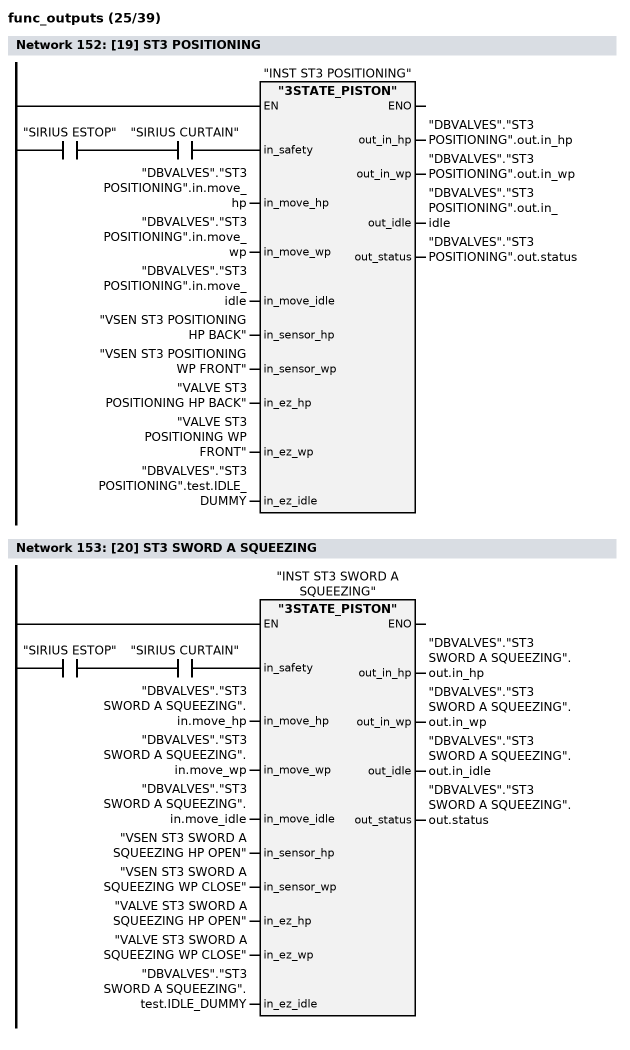
   RUNG wire#powerrail
      "INST ST3 POSITIONING"(in_safety := wire#w1, in_move_hp := "DBVALVES"."ST3 POSITIONING".in.move_hp, in_move_wp := "DBVALVES"."ST3 POSITIONING".in.move_wp, in_move_idle := "DBVALVES"."ST3 POSITIONING".in.move_idle, in_sensor_hp := "VSEN ST3 POSITIONING HP BACK", in_sensor_wp := "VSEN ST3 POSITIONING WP FRONT", in_ez_hp := "VALVE ST3 POSITIONING HP BACK", in_ez_wp := "VALVE ST3 POSITIONING WP FRONT", in_ez_idle := "DBVALVES"."ST3 POSITIONING".test.IDLE_DUMMY, out_in_hp => "DBVALVES"."ST3 POSITIONING".out.in_hp, out_in_wp => "DBVALVES"."ST3 POSITIONING".out.in_wp, out_idle => "DBVALVES"."ST3 POSITIONING".out.in_idle, out_status => "DBVALVES"."ST3 POSITIONING".out.status)
   END_RUNG
   RUNG wire#powerrail
      Contact( "SIRIUS ESTOP" )
      Contact( "SIRIUS CURTAIN" )
   END_RUNG wire#w1
   // the same network as SCL:
   "INST ST3 POSITIONING"(in_safety := "SIRIUS ESTOP" AND "SIRIUS CURTAIN",   // "3STATE_PISTON"
                          in_move_hp := "DBVALVES"."ST3 POSITIONING".in.move_hp,
                          in_move_wp := "DBVALVES"."ST3 POSITIONING".in.move_wp,
                          in_move_idle := "DBVALVES"."ST3 POSITIONING".in.move_idle,
                          in_sensor_hp := "VSEN ST3 POSITIONING HP BACK",
                          in_sensor_wp := "VSEN ST3 POSITIONING WP FRONT",
                          in_ez_hp := "VALVE ST3 POSITIONING HP BACK",
                          in_ez_wp := "VALVE ST3 POSITIONING WP FRONT",
                          in_ez_idle := "DBVALVES"."ST3 POSITIONING".test.IDLE_DUMMY,
                          out_in_hp => "DBVALVES"."ST3 POSITIONING".out.in_hp,
                          out_in_wp => "DBVALVES"."ST3 POSITIONING".out.in_wp,
                          out_idle => "DBVALVES"."ST3 POSITIONING".out.in_idle,
                          out_status => "DBVALVES"."ST3 POSITIONING".out.status);
END_REGION

REGION Network 153: [20] ST3 SWORD A SQUEEZING
   RUNG wire#powerrail
      "INST ST3 SWORD A SQUEEZING"(in_safety := wire#w1, in_move_hp := "DBVALVES"."ST3 SWORD A SQUEEZING".in.move_hp, in_move_wp := "DBVALVES"."ST3 SWORD A SQUEEZING".in.move_wp, in_move_idle := "DBVALVES"."ST3 SWORD A SQUEEZING".in.move_idle, in_sensor_hp := "VSEN ST3 SWORD A SQUEEZING HP OPEN", in_sensor_wp := "VSEN ST3 SWORD A SQUEEZING WP CLOSE", in_ez_hp := "VALVE ST3 SWORD A SQUEEZING HP OPEN", in_ez_wp := "VALVE ST3 SWORD A SQUEEZING WP CLOSE", in_ez_idle := "DBVALVES"."ST3 SWORD A SQUEEZING".test.IDLE_DUMMY, out_in_hp => "DBVALVES"."ST3 SWORD A SQUEEZING".out.in_hp, out_in_wp => "DBVALVES"."ST3 SWORD A SQUEEZING".out.in_wp, out_idle => "DBVALVES"."ST3 SWORD A SQUEEZING".out.in_idle, out_status => "DBVALVES"."ST3 SWORD A SQUEEZING".out.status)
   END_RUNG
   RUNG wire#powerrail
      Contact( "SIRIUS ESTOP" )
      Contact( "SIRIUS CURTAIN" )
   END_RUNG wire#w1
   // the same network as SCL:
   "INST ST3 SWORD A SQUEEZING"(in_safety := "SIRIUS ESTOP" AND "SIRIUS CURTAIN",   // "3STATE_PISTON"
                           in_move_hp := "DBVALVES"."ST3 SWORD A SQUEEZING".in.move_hp,
                           in_move_wp := "DBVALVES"."ST3 SWORD A SQUEEZING".in.move_wp,
                           in_move_idle := "DBVALVES"."ST3 SWORD A SQUEEZING".in.move_idle,
                           in_sensor_hp := "VSEN ST3 SWORD A SQUEEZING HP OPEN",
                           in_sensor_wp := "VSEN ST3 SWORD A SQUEEZING WP CLOSE",
                           in_ez_hp := "VALVE ST3 SWORD A SQUEEZING HP OPEN",
                           in_ez_wp := "VALVE ST3 SWORD A SQUEEZING WP CLOSE",
                           in_ez_idle := "DBVALVES"."ST3 SWORD A SQUEEZING".test.IDLE_DUMMY,
                           out_in_hp => "DBVALVES"."ST3 SWORD A SQUEEZING".out.in_hp,
                           out_in_wp => "DBVALVES"."ST3 SWORD A SQUEEZING".out.in_wp,
                           out_idle => "DBVALVES"."ST3 SWORD A SQUEEZING".out.in_idle,
                           out_status => "DBVALVES"."ST3 SWORD A SQUEEZING".out.status);
END_REGION

REGION Network 154: [21] ST3 SWORD A SPREADING
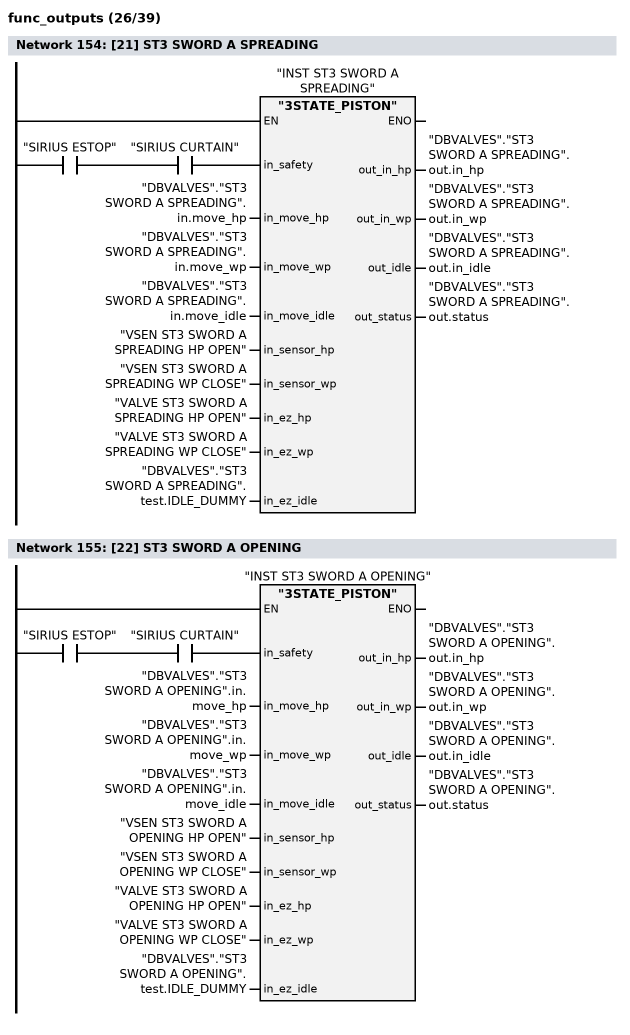
   RUNG wire#powerrail
      "INST ST3 SWORD A SPREADING"(in_safety := wire#w1, in_move_hp := "DBVALVES"."ST3 SWORD A SPREADING".in.move_hp, in_move_wp := "DBVALVES"."ST3 SWORD A SPREADING".in.move_wp, in_move_idle := "DBVALVES"."ST3 SWORD A SPREADING".in.move_idle, in_sensor_hp := "VSEN ST3 SWORD A SPREADING HP OPEN", in_sensor_wp := "VSEN ST3 SWORD A SPREADING WP CLOSE", in_ez_hp := "VALVE ST3 SWORD A SPREADING HP OPEN", in_ez_wp := "VALVE ST3 SWORD A SPREADING WP CLOSE", in_ez_idle := "DBVALVES"."ST3 SWORD A SPREADING".test.IDLE_DUMMY, out_in_hp => "DBVALVES"."ST3 SWORD A SPREADING".out.in_hp, out_in_wp => "DBVALVES"."ST3 SWORD A SPREADING".out.in_wp, out_idle => "DBVALVES"."ST3 SWORD A SPREADING".out.in_idle, out_status => "DBVALVES"."ST3 SWORD A SPREADING".out.status)
   END_RUNG
   RUNG wire#powerrail
      Contact( "SIRIUS ESTOP" )
      Contact( "SIRIUS CURTAIN" )
   END_RUNG wire#w1
   // the same network as SCL:
   "INST ST3 SWORD A SPREADING"(in_safety := "SIRIUS ESTOP" AND "SIRIUS CURTAIN",   // "3STATE_PISTON"
                           in_move_hp := "DBVALVES"."ST3 SWORD A SPREADING".in.move_hp,
                           in_move_wp := "DBVALVES"."ST3 SWORD A SPREADING".in.move_wp,
                           in_move_idle := "DBVALVES"."ST3 SWORD A SPREADING".in.move_idle,
                           in_sensor_hp := "VSEN ST3 SWORD A SPREADING HP OPEN",
                           in_sensor_wp := "VSEN ST3 SWORD A SPREADING WP CLOSE",
                           in_ez_hp := "VALVE ST3 SWORD A SPREADING HP OPEN",
                           in_ez_wp := "VALVE ST3 SWORD A SPREADING WP CLOSE",
                           in_ez_idle := "DBVALVES"."ST3 SWORD A SPREADING".test.IDLE_DUMMY,
                           out_in_hp => "DBVALVES"."ST3 SWORD A SPREADING".out.in_hp,
                           out_in_wp => "DBVALVES"."ST3 SWORD A SPREADING".out.in_wp,
                           out_idle => "DBVALVES"."ST3 SWORD A SPREADING".out.in_idle,
                           out_status => "DBVALVES"."ST3 SWORD A SPREADING".out.status);
END_REGION

REGION Network 155: [22] ST3 SWORD A OPENING
   RUNG wire#powerrail
      "INST ST3 SWORD A OPENING"(in_safety := wire#w1, in_move_hp := "DBVALVES"."ST3 SWORD A OPENING".in.move_hp, in_move_wp := "DBVALVES"."ST3 SWORD A OPENING".in.move_wp, in_move_idle := "DBVALVES"."ST3 SWORD A OPENING".in.move_idle, in_sensor_hp := "VSEN ST3 SWORD A OPENING HP OPEN", in_sensor_wp := "VSEN ST3 SWORD A OPENING WP CLOSE", in_ez_hp := "VALVE ST3 SWORD A OPENING HP OPEN", in_ez_wp := "VALVE ST3 SWORD A OPENING WP CLOSE", in_ez_idle := "DBVALVES"."ST3 SWORD A OPENING".test.IDLE_DUMMY, out_in_hp => "DBVALVES"."ST3 SWORD A OPENING".out.in_hp, out_in_wp => "DBVALVES"."ST3 SWORD A OPENING".out.in_wp, out_idle => "DBVALVES"."ST3 SWORD A OPENING".out.in_idle, out_status => "DBVALVES"."ST3 SWORD A OPENING".out.status)
   END_RUNG
   RUNG wire#powerrail
      Contact( "SIRIUS ESTOP" )
      Contact( "SIRIUS CURTAIN" )
   END_RUNG wire#w1
   // the same network as SCL:
   "INST ST3 SWORD A OPENING"(in_safety := "SIRIUS ESTOP" AND "SIRIUS CURTAIN",   // "3STATE_PISTON"
                           in_move_hp := "DBVALVES"."ST3 SWORD A OPENING".in.move_hp,
                           in_move_wp := "DBVALVES"."ST3 SWORD A OPENING".in.move_wp,
                           in_move_idle := "DBVALVES"."ST3 SWORD A OPENING".in.move_idle,
                           in_sensor_hp := "VSEN ST3 SWORD A OPENING HP OPEN",
                           in_sensor_wp := "VSEN ST3 SWORD A OPENING WP CLOSE",
                           in_ez_hp := "VALVE ST3 SWORD A OPENING HP OPEN",
                           in_ez_wp := "VALVE ST3 SWORD A OPENING WP CLOSE",
                           in_ez_idle := "DBVALVES"."ST3 SWORD A OPENING".test.IDLE_DUMMY,
                           out_in_hp => "DBVALVES"."ST3 SWORD A OPENING".out.in_hp,
                           out_in_wp => "DBVALVES"."ST3 SWORD A OPENING".out.in_wp,
                           out_idle => "DBVALVES"."ST3 SWORD A OPENING".out.in_idle,
                           out_status => "DBVALVES"."ST3 SWORD A OPENING".out.status);
END_REGION

REGION Network 156: [23] ST3 SWORD B SQUEEZING
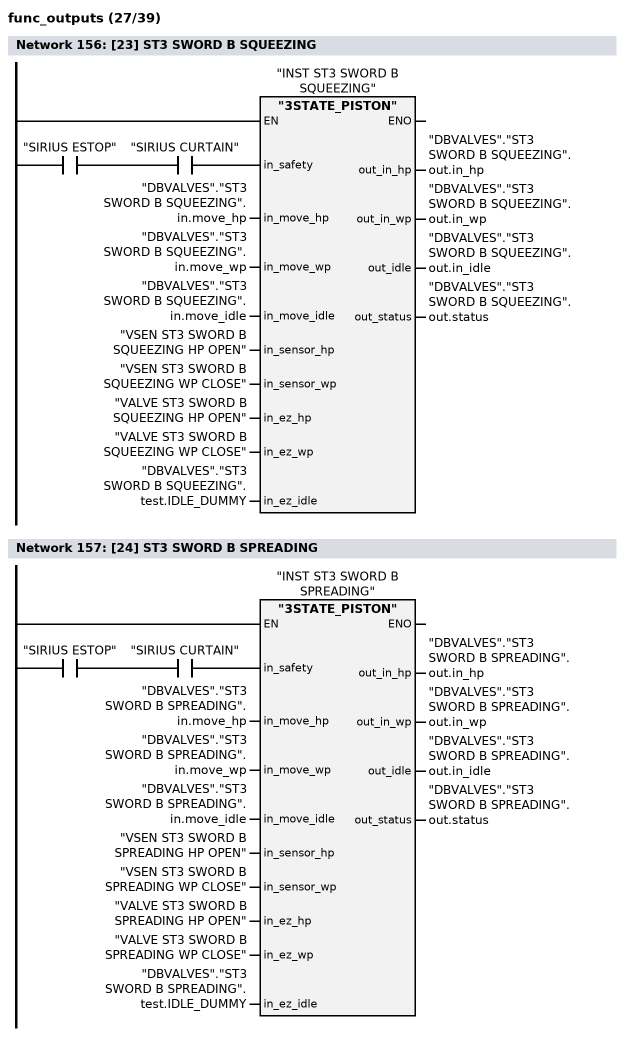
   RUNG wire#powerrail
      "INST ST3 SWORD B SQUEEZING"(in_safety := wire#w1, in_move_hp := "DBVALVES"."ST3 SWORD B SQUEEZING".in.move_hp, in_move_wp := "DBVALVES"."ST3 SWORD B SQUEEZING".in.move_wp, in_move_idle := "DBVALVES"."ST3 SWORD B SQUEEZING".in.move_idle, in_sensor_hp := "VSEN ST3 SWORD B SQUEEZING HP OPEN", in_sensor_wp := "VSEN ST3 SWORD B SQUEEZING WP CLOSE", in_ez_hp := "VALVE ST3 SWORD B SQUEEZING HP OPEN", in_ez_wp := "VALVE ST3 SWORD B SQUEEZING WP CLOSE", in_ez_idle := "DBVALVES"."ST3 SWORD B SQUEEZING".test.IDLE_DUMMY, out_in_hp => "DBVALVES"."ST3 SWORD B SQUEEZING".out.in_hp, out_in_wp => "DBVALVES"."ST3 SWORD B SQUEEZING".out.in_wp, out_idle => "DBVALVES"."ST3 SWORD B SQUEEZING".out.in_idle, out_status => "DBVALVES"."ST3 SWORD B SQUEEZING".out.status)
   END_RUNG
   RUNG wire#powerrail
      Contact( "SIRIUS ESTOP" )
      Contact( "SIRIUS CURTAIN" )
   END_RUNG wire#w1
   // the same network as SCL:
   "INST ST3 SWORD B SQUEEZING"(in_safety := "SIRIUS ESTOP" AND "SIRIUS CURTAIN",   // "3STATE_PISTON"
                           in_move_hp := "DBVALVES"."ST3 SWORD B SQUEEZING".in.move_hp,
                           in_move_wp := "DBVALVES"."ST3 SWORD B SQUEEZING".in.move_wp,
                           in_move_idle := "DBVALVES"."ST3 SWORD B SQUEEZING".in.move_idle,
                           in_sensor_hp := "VSEN ST3 SWORD B SQUEEZING HP OPEN",
                           in_sensor_wp := "VSEN ST3 SWORD B SQUEEZING WP CLOSE",
                           in_ez_hp := "VALVE ST3 SWORD B SQUEEZING HP OPEN",
                           in_ez_wp := "VALVE ST3 SWORD B SQUEEZING WP CLOSE",
                           in_ez_idle := "DBVALVES"."ST3 SWORD B SQUEEZING".test.IDLE_DUMMY,
                           out_in_hp => "DBVALVES"."ST3 SWORD B SQUEEZING".out.in_hp,
                           out_in_wp => "DBVALVES"."ST3 SWORD B SQUEEZING".out.in_wp,
                           out_idle => "DBVALVES"."ST3 SWORD B SQUEEZING".out.in_idle,
                           out_status => "DBVALVES"."ST3 SWORD B SQUEEZING".out.status);
END_REGION

REGION Network 157: [24] ST3 SWORD B SPREADING
   RUNG wire#powerrail
      "INST ST3 SWORD B SPREADING"(in_safety := wire#w1, in_move_hp := "DBVALVES"."ST3 SWORD B SPREADING".in.move_hp, in_move_wp := "DBVALVES"."ST3 SWORD B SPREADING".in.move_wp, in_move_idle := "DBVALVES"."ST3 SWORD B SPREADING".in.move_idle, in_sensor_hp := "VSEN ST3 SWORD B SPREADING HP OPEN", in_sensor_wp := "VSEN ST3 SWORD B SPREADING WP CLOSE", in_ez_hp := "VALVE ST3 SWORD B SPREADING HP OPEN", in_ez_wp := "VALVE ST3 SWORD B SPREADING WP CLOSE", in_ez_idle := "DBVALVES"."ST3 SWORD B SPREADING".test.IDLE_DUMMY, out_in_hp => "DBVALVES"."ST3 SWORD B SPREADING".out.in_hp, out_in_wp => "DBVALVES"."ST3 SWORD B SPREADING".out.in_wp, out_idle => "DBVALVES"."ST3 SWORD B SPREADING".out.in_idle, out_status => "DBVALVES"."ST3 SWORD B SPREADING".out.status)
   END_RUNG
   RUNG wire#powerrail
      Contact( "SIRIUS ESTOP" )
      Contact( "SIRIUS CURTAIN" )
   END_RUNG wire#w1
   // the same network as SCL:
   "INST ST3 SWORD B SPREADING"(in_safety := "SIRIUS ESTOP" AND "SIRIUS CURTAIN",   // "3STATE_PISTON"
                           in_move_hp := "DBVALVES"."ST3 SWORD B SPREADING".in.move_hp,
                           in_move_wp := "DBVALVES"."ST3 SWORD B SPREADING".in.move_wp,
                           in_move_idle := "DBVALVES"."ST3 SWORD B SPREADING".in.move_idle,
                           in_sensor_hp := "VSEN ST3 SWORD B SPREADING HP OPEN",
                           in_sensor_wp := "VSEN ST3 SWORD B SPREADING WP CLOSE",
                           in_ez_hp := "VALVE ST3 SWORD B SPREADING HP OPEN",
                           in_ez_wp := "VALVE ST3 SWORD B SPREADING WP CLOSE",
                           in_ez_idle := "DBVALVES"."ST3 SWORD B SPREADING".test.IDLE_DUMMY,
                           out_in_hp => "DBVALVES"."ST3 SWORD B SPREADING".out.in_hp,
                           out_in_wp => "DBVALVES"."ST3 SWORD B SPREADING".out.in_wp,
                           out_idle => "DBVALVES"."ST3 SWORD B SPREADING".out.in_idle,
                           out_status => "DBVALVES"."ST3 SWORD B SPREADING".out.status);
END_REGION

REGION Network 158: [25] ST3 SWORD B OPENING
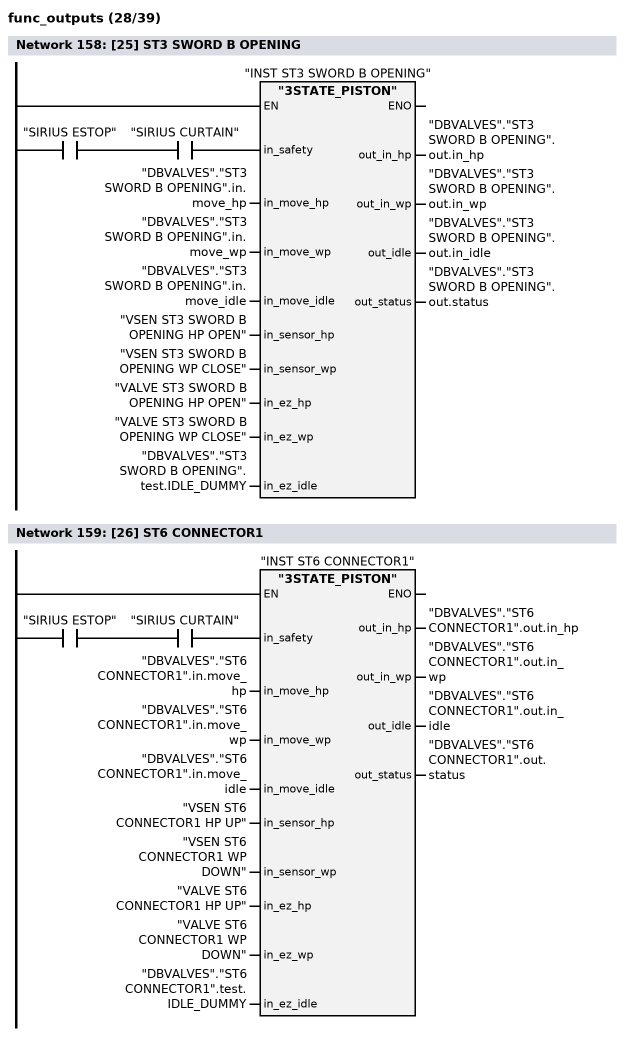
   RUNG wire#powerrail
      "INST ST3 SWORD B OPENING"(in_safety := wire#w1, in_move_hp := "DBVALVES"."ST3 SWORD B OPENING".in.move_hp, in_move_wp := "DBVALVES"."ST3 SWORD B OPENING".in.move_wp, in_move_idle := "DBVALVES"."ST3 SWORD B OPENING".in.move_idle, in_sensor_hp := "VSEN ST3 SWORD B OPENING HP OPEN", in_sensor_wp := "VSEN ST3 SWORD B OPENING WP CLOSE", in_ez_hp := "VALVE ST3 SWORD B OPENING HP OPEN", in_ez_wp := "VALVE ST3 SWORD B OPENING WP CLOSE", in_ez_idle := "DBVALVES"."ST3 SWORD B OPENING".test.IDLE_DUMMY, out_in_hp => "DBVALVES"."ST3 SWORD B OPENING".out.in_hp, out_in_wp => "DBVALVES"."ST3 SWORD B OPENING".out.in_wp, out_idle => "DBVALVES"."ST3 SWORD B OPENING".out.in_idle, out_status => "DBVALVES"."ST3 SWORD B OPENING".out.status)
   END_RUNG
   RUNG wire#powerrail
      Contact( "SIRIUS ESTOP" )
      Contact( "SIRIUS CURTAIN" )
   END_RUNG wire#w1
   // the same network as SCL:
   "INST ST3 SWORD B OPENING"(in_safety := "SIRIUS ESTOP" AND "SIRIUS CURTAIN",   // "3STATE_PISTON"
                           in_move_hp := "DBVALVES"."ST3 SWORD B OPENING".in.move_hp,
                           in_move_wp := "DBVALVES"."ST3 SWORD B OPENING".in.move_wp,
                           in_move_idle := "DBVALVES"."ST3 SWORD B OPENING".in.move_idle,
                           in_sensor_hp := "VSEN ST3 SWORD B OPENING HP OPEN",
                           in_sensor_wp := "VSEN ST3 SWORD B OPENING WP CLOSE",
                           in_ez_hp := "VALVE ST3 SWORD B OPENING HP OPEN",
                           in_ez_wp := "VALVE ST3 SWORD B OPENING WP CLOSE",
                           in_ez_idle := "DBVALVES"."ST3 SWORD B OPENING".test.IDLE_DUMMY,
                           out_in_hp => "DBVALVES"."ST3 SWORD B OPENING".out.in_hp,
                           out_in_wp => "DBVALVES"."ST3 SWORD B OPENING".out.in_wp,
                           out_idle => "DBVALVES"."ST3 SWORD B OPENING".out.in_idle,
                           out_status => "DBVALVES"."ST3 SWORD B OPENING".out.status);
END_REGION

REGION Network 159: [26] ST6 CONNECTOR1
   RUNG wire#powerrail
      "INST ST6 CONNECTOR1"(in_safety := wire#w1, in_move_hp := "DBVALVES"."ST6 CONNECTOR1".in.move_hp, in_move_wp := "DBVALVES"."ST6 CONNECTOR1".in.move_wp, in_move_idle := "DBVALVES"."ST6 CONNECTOR1".in.move_idle, in_sensor_hp := "VSEN ST6 CONNECTOR1 HP UP", in_sensor_wp := "VSEN ST6 CONNECTOR1 WP DOWN", in_ez_hp := "VALVE ST6 CONNECTOR1 HP UP", in_ez_wp := "VALVE ST6 CONNECTOR1 WP DOWN", in_ez_idle := "DBVALVES"."ST6 CONNECTOR1".test.IDLE_DUMMY, out_in_hp => "DBVALVES"."ST6 CONNECTOR1".out.in_hp, out_in_wp => "DBVALVES"."ST6 CONNECTOR1".out.in_wp, out_idle => "DBVALVES"."ST6 CONNECTOR1".out.in_idle, out_status => "DBVALVES"."ST6 CONNECTOR1".out.status)
   END_RUNG
   RUNG wire#powerrail
      Contact( "SIRIUS ESTOP" )
      Contact( "SIRIUS CURTAIN" )
   END_RUNG wire#w1
   // the same network as SCL:
   "INST ST6 CONNECTOR1"(in_safety := "SIRIUS ESTOP" AND "SIRIUS CURTAIN",   // "3STATE_PISTON"
                         in_move_hp := "DBVALVES"."ST6 CONNECTOR1".in.move_hp,
                         in_move_wp := "DBVALVES"."ST6 CONNECTOR1".in.move_wp,
                         in_move_idle := "DBVALVES"."ST6 CONNECTOR1".in.move_idle,
                         in_sensor_hp := "VSEN ST6 CONNECTOR1 HP UP",
                         in_sensor_wp := "VSEN ST6 CONNECTOR1 WP DOWN",
                         in_ez_hp := "VALVE ST6 CONNECTOR1 HP UP",
                         in_ez_wp := "VALVE ST6 CONNECTOR1 WP DOWN",
                         in_ez_idle := "DBVALVES"."ST6 CONNECTOR1".test.IDLE_DUMMY,
                         out_in_hp => "DBVALVES"."ST6 CONNECTOR1".out.in_hp,
                         out_in_wp => "DBVALVES"."ST6 CONNECTOR1".out.in_wp,
                         out_idle => "DBVALVES"."ST6 CONNECTOR1".out.in_idle,
                         out_status => "DBVALVES"."ST6 CONNECTOR1".out.status);
END_REGION

REGION Network 160: [27] ST6 CONNECTOR2
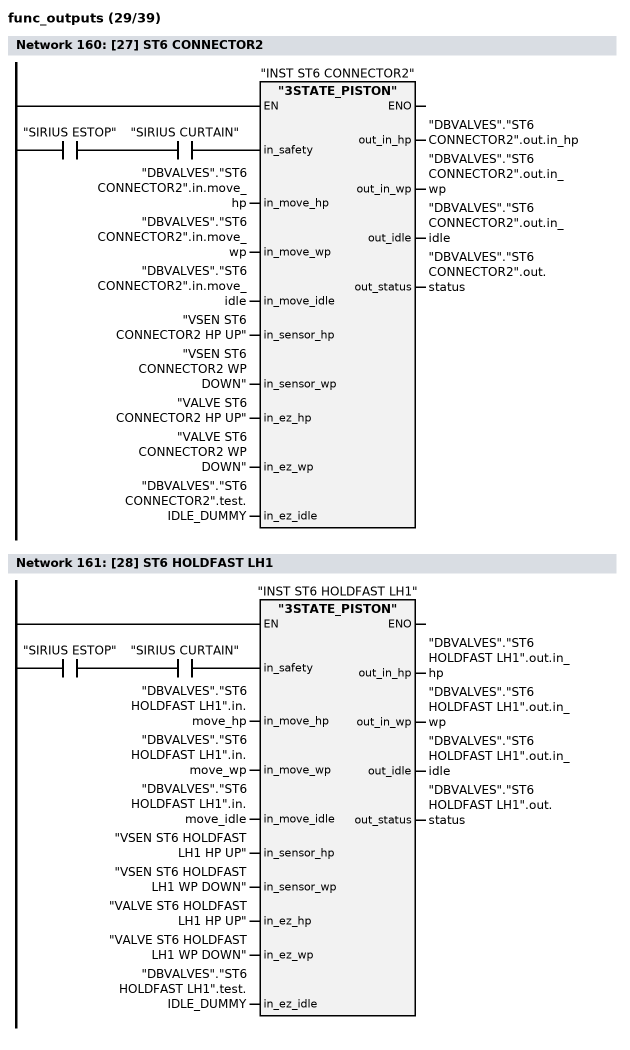
   RUNG wire#powerrail
      "INST ST6 CONNECTOR2"(in_safety := wire#w1, in_move_hp := "DBVALVES"."ST6 CONNECTOR2".in.move_hp, in_move_wp := "DBVALVES"."ST6 CONNECTOR2".in.move_wp, in_move_idle := "DBVALVES"."ST6 CONNECTOR2".in.move_idle, in_sensor_hp := "VSEN ST6 CONNECTOR2 HP UP", in_sensor_wp := "VSEN ST6 CONNECTOR2 WP DOWN", in_ez_hp := "VALVE ST6 CONNECTOR2 HP UP", in_ez_wp := "VALVE ST6 CONNECTOR2 WP DOWN", in_ez_idle := "DBVALVES"."ST6 CONNECTOR2".test.IDLE_DUMMY, out_in_hp => "DBVALVES"."ST6 CONNECTOR2".out.in_hp, out_in_wp => "DBVALVES"."ST6 CONNECTOR2".out.in_wp, out_idle => "DBVALVES"."ST6 CONNECTOR2".out.in_idle, out_status => "DBVALVES"."ST6 CONNECTOR2".out.status)
   END_RUNG
   RUNG wire#powerrail
      Contact( "SIRIUS ESTOP" )
      Contact( "SIRIUS CURTAIN" )
   END_RUNG wire#w1
   // the same network as SCL:
   "INST ST6 CONNECTOR2"(in_safety := "SIRIUS ESTOP" AND "SIRIUS CURTAIN",   // "3STATE_PISTON"
                         in_move_hp := "DBVALVES"."ST6 CONNECTOR2".in.move_hp,
                         in_move_wp := "DBVALVES"."ST6 CONNECTOR2".in.move_wp,
                         in_move_idle := "DBVALVES"."ST6 CONNECTOR2".in.move_idle,
                         in_sensor_hp := "VSEN ST6 CONNECTOR2 HP UP",
                         in_sensor_wp := "VSEN ST6 CONNECTOR2 WP DOWN",
                         in_ez_hp := "VALVE ST6 CONNECTOR2 HP UP",
                         in_ez_wp := "VALVE ST6 CONNECTOR2 WP DOWN",
                         in_ez_idle := "DBVALVES"."ST6 CONNECTOR2".test.IDLE_DUMMY,
                         out_in_hp => "DBVALVES"."ST6 CONNECTOR2".out.in_hp,
                         out_in_wp => "DBVALVES"."ST6 CONNECTOR2".out.in_wp,
                         out_idle => "DBVALVES"."ST6 CONNECTOR2".out.in_idle,
                         out_status => "DBVALVES"."ST6 CONNECTOR2".out.status);
END_REGION

REGION Network 161: [28] ST6 HOLDFAST LH1
   RUNG wire#powerrail
      "INST ST6 HOLDFAST LH1"(in_safety := wire#w1, in_move_hp := "DBVALVES"."ST6 HOLDFAST LH1".in.move_hp, in_move_wp := "DBVALVES"."ST6 HOLDFAST LH1".in.move_wp, in_move_idle := "DBVALVES"."ST6 HOLDFAST LH1".in.move_idle, in_sensor_hp := "VSEN ST6 HOLDFAST LH1 HP UP", in_sensor_wp := "VSEN ST6 HOLDFAST LH1 WP DOWN", in_ez_hp := "VALVE ST6 HOLDFAST LH1 HP UP", in_ez_wp := "VALVE ST6 HOLDFAST LH1 WP DOWN", in_ez_idle := "DBVALVES"."ST6 HOLDFAST LH1".test.IDLE_DUMMY, out_in_hp => "DBVALVES"."ST6 HOLDFAST LH1".out.in_hp, out_in_wp => "DBVALVES"."ST6 HOLDFAST LH1".out.in_wp, out_idle => "DBVALVES"."ST6 HOLDFAST LH1".out.in_idle, out_status => "DBVALVES"."ST6 HOLDFAST LH1".out.status)
   END_RUNG
   RUNG wire#powerrail
      Contact( "SIRIUS ESTOP" )
      Contact( "SIRIUS CURTAIN" )
   END_RUNG wire#w1
   // the same network as SCL:
   "INST ST6 HOLDFAST LH1"(in_safety := "SIRIUS ESTOP" AND "SIRIUS CURTAIN",   // "3STATE_PISTON"
                           in_move_hp := "DBVALVES"."ST6 HOLDFAST LH1".in.move_hp,
                           in_move_wp := "DBVALVES"."ST6 HOLDFAST LH1".in.move_wp,
                           in_move_idle := "DBVALVES"."ST6 HOLDFAST LH1".in.move_idle,
                           in_sensor_hp := "VSEN ST6 HOLDFAST LH1 HP UP",
                           in_sensor_wp := "VSEN ST6 HOLDFAST LH1 WP DOWN",
                           in_ez_hp := "VALVE ST6 HOLDFAST LH1 HP UP",
                           in_ez_wp := "VALVE ST6 HOLDFAST LH1 WP DOWN",
                           in_ez_idle := "DBVALVES"."ST6 HOLDFAST LH1".test.IDLE_DUMMY,
                           out_in_hp => "DBVALVES"."ST6 HOLDFAST LH1".out.in_hp,
                           out_in_wp => "DBVALVES"."ST6 HOLDFAST LH1".out.in_wp,
                           out_idle => "DBVALVES"."ST6 HOLDFAST LH1".out.in_idle,
                           out_status => "DBVALVES"."ST6 HOLDFAST LH1".out.status);
END_REGION

REGION Network 162: [29] ST6 HOLDFAST LH2
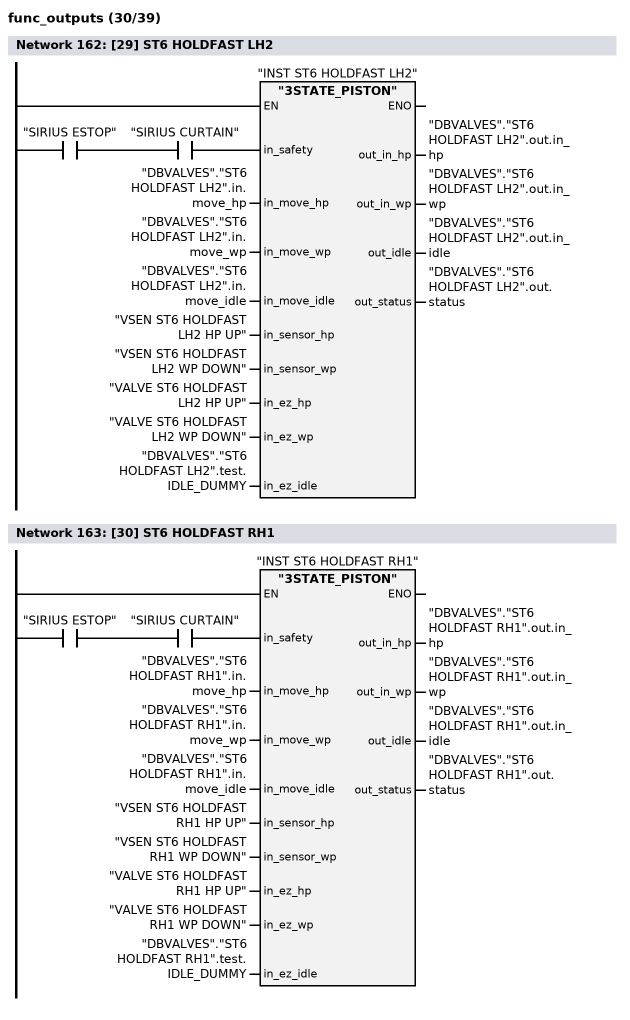
   RUNG wire#powerrail
      "INST ST6 HOLDFAST LH2"(in_safety := wire#w1, in_move_hp := "DBVALVES"."ST6 HOLDFAST LH2".in.move_hp, in_move_wp := "DBVALVES"."ST6 HOLDFAST LH2".in.move_wp, in_move_idle := "DBVALVES"."ST6 HOLDFAST LH2".in.move_idle, in_sensor_hp := "VSEN ST6 HOLDFAST LH2 HP UP", in_sensor_wp := "VSEN ST6 HOLDFAST LH2 WP DOWN", in_ez_hp := "VALVE ST6 HOLDFAST LH2 HP UP", in_ez_wp := "VALVE ST6 HOLDFAST LH2 WP DOWN", in_ez_idle := "DBVALVES"."ST6 HOLDFAST LH2".test.IDLE_DUMMY, out_in_hp => "DBVALVES"."ST6 HOLDFAST LH2".out.in_hp, out_in_wp => "DBVALVES"."ST6 HOLDFAST LH2".out.in_wp, out_idle => "DBVALVES"."ST6 HOLDFAST LH2".out.in_idle, out_status => "DBVALVES"."ST6 HOLDFAST LH2".out.status)
   END_RUNG
   RUNG wire#powerrail
      Contact( "SIRIUS ESTOP" )
      Contact( "SIRIUS CURTAIN" )
   END_RUNG wire#w1
   // the same network as SCL:
   "INST ST6 HOLDFAST LH2"(in_safety := "SIRIUS ESTOP" AND "SIRIUS CURTAIN",   // "3STATE_PISTON"
                           in_move_hp := "DBVALVES"."ST6 HOLDFAST LH2".in.move_hp,
                           in_move_wp := "DBVALVES"."ST6 HOLDFAST LH2".in.move_wp,
                           in_move_idle := "DBVALVES"."ST6 HOLDFAST LH2".in.move_idle,
                           in_sensor_hp := "VSEN ST6 HOLDFAST LH2 HP UP",
                           in_sensor_wp := "VSEN ST6 HOLDFAST LH2 WP DOWN",
                           in_ez_hp := "VALVE ST6 HOLDFAST LH2 HP UP",
                           in_ez_wp := "VALVE ST6 HOLDFAST LH2 WP DOWN",
                           in_ez_idle := "DBVALVES"."ST6 HOLDFAST LH2".test.IDLE_DUMMY,
                           out_in_hp => "DBVALVES"."ST6 HOLDFAST LH2".out.in_hp,
                           out_in_wp => "DBVALVES"."ST6 HOLDFAST LH2".out.in_wp,
                           out_idle => "DBVALVES"."ST6 HOLDFAST LH2".out.in_idle,
                           out_status => "DBVALVES"."ST6 HOLDFAST LH2".out.status);
END_REGION

REGION Network 163: [30] ST6 HOLDFAST RH1
   RUNG wire#powerrail
      "INST ST6 HOLDFAST RH1"(in_safety := wire#w1, in_move_hp := "DBVALVES"."ST6 HOLDFAST RH1".in.move_hp, in_move_wp := "DBVALVES"."ST6 HOLDFAST RH1".in.move_wp, in_move_idle := "DBVALVES"."ST6 HOLDFAST RH1".in.move_idle, in_sensor_hp := "VSEN ST6 HOLDFAST RH1 HP UP", in_sensor_wp := "VSEN ST6 HOLDFAST RH1 WP DOWN", in_ez_hp := "VALVE ST6 HOLDFAST RH1 HP UP", in_ez_wp := "VALVE ST6 HOLDFAST RH1 WP DOWN", in_ez_idle := "DBVALVES"."ST6 HOLDFAST RH1".test.IDLE_DUMMY, out_in_hp => "DBVALVES"."ST6 HOLDFAST RH1".out.in_hp, out_in_wp => "DBVALVES"."ST6 HOLDFAST RH1".out.in_wp, out_idle => "DBVALVES"."ST6 HOLDFAST RH1".out.in_idle, out_status => "DBVALVES"."ST6 HOLDFAST RH1".out.status)
   END_RUNG
   RUNG wire#powerrail
      Contact( "SIRIUS ESTOP" )
      Contact( "SIRIUS CURTAIN" )
   END_RUNG wire#w1
   // the same network as SCL:
   "INST ST6 HOLDFAST RH1"(in_safety := "SIRIUS ESTOP" AND "SIRIUS CURTAIN",   // "3STATE_PISTON"
                           in_move_hp := "DBVALVES"."ST6 HOLDFAST RH1".in.move_hp,
                           in_move_wp := "DBVALVES"."ST6 HOLDFAST RH1".in.move_wp,
                           in_move_idle := "DBVALVES"."ST6 HOLDFAST RH1".in.move_idle,
                           in_sensor_hp := "VSEN ST6 HOLDFAST RH1 HP UP",
                           in_sensor_wp := "VSEN ST6 HOLDFAST RH1 WP DOWN",
                           in_ez_hp := "VALVE ST6 HOLDFAST RH1 HP UP",
                           in_ez_wp := "VALVE ST6 HOLDFAST RH1 WP DOWN",
                           in_ez_idle := "DBVALVES"."ST6 HOLDFAST RH1".test.IDLE_DUMMY,
                           out_in_hp => "DBVALVES"."ST6 HOLDFAST RH1".out.in_hp,
                           out_in_wp => "DBVALVES"."ST6 HOLDFAST RH1".out.in_wp,
                           out_idle => "DBVALVES"."ST6 HOLDFAST RH1".out.in_idle,
                           out_status => "DBVALVES"."ST6 HOLDFAST RH1".out.status);
END_REGION

REGION Network 164: [31] ST6 HOLDFAST RH2
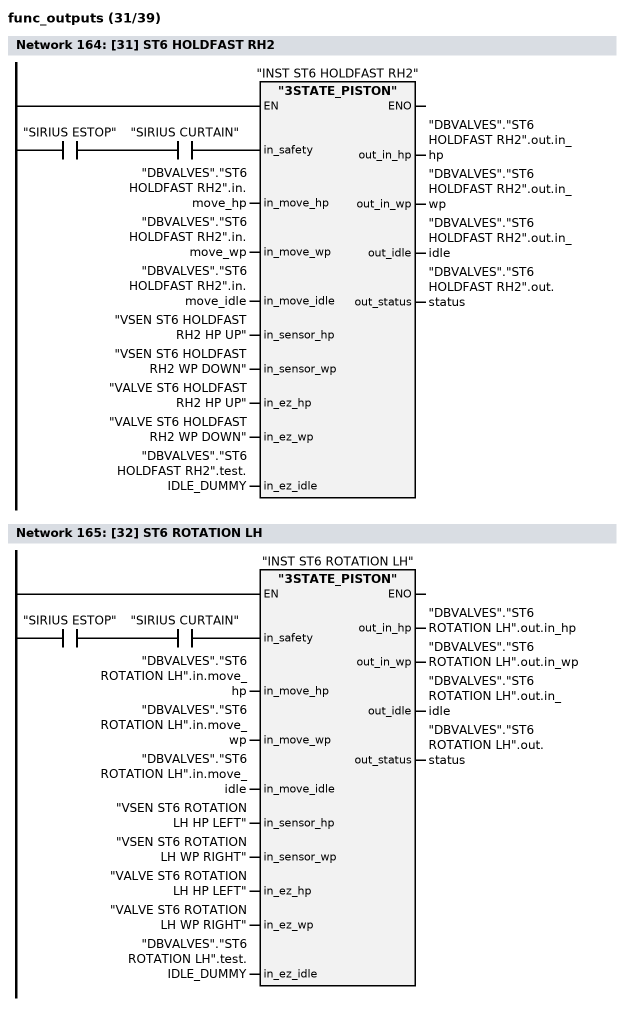
   RUNG wire#powerrail
      "INST ST6 HOLDFAST RH2"(in_safety := wire#w1, in_move_hp := "DBVALVES"."ST6 HOLDFAST RH2".in.move_hp, in_move_wp := "DBVALVES"."ST6 HOLDFAST RH2".in.move_wp, in_move_idle := "DBVALVES"."ST6 HOLDFAST RH2".in.move_idle, in_sensor_hp := "VSEN ST6 HOLDFAST RH2 HP UP", in_sensor_wp := "VSEN ST6 HOLDFAST RH2 WP DOWN", in_ez_hp := "VALVE ST6 HOLDFAST RH2 HP UP", in_ez_wp := "VALVE ST6 HOLDFAST RH2 WP DOWN", in_ez_idle := "DBVALVES"."ST6 HOLDFAST RH2".test.IDLE_DUMMY, out_in_hp => "DBVALVES"."ST6 HOLDFAST RH2".out.in_hp, out_in_wp => "DBVALVES"."ST6 HOLDFAST RH2".out.in_wp, out_idle => "DBVALVES"."ST6 HOLDFAST RH2".out.in_idle, out_status => "DBVALVES"."ST6 HOLDFAST RH2".out.status)
   END_RUNG
   RUNG wire#powerrail
      Contact( "SIRIUS ESTOP" )
      Contact( "SIRIUS CURTAIN" )
   END_RUNG wire#w1
   // the same network as SCL:
   "INST ST6 HOLDFAST RH2"(in_safety := "SIRIUS ESTOP" AND "SIRIUS CURTAIN",   // "3STATE_PISTON"
                           in_move_hp := "DBVALVES"."ST6 HOLDFAST RH2".in.move_hp,
                           in_move_wp := "DBVALVES"."ST6 HOLDFAST RH2".in.move_wp,
                           in_move_idle := "DBVALVES"."ST6 HOLDFAST RH2".in.move_idle,
                           in_sensor_hp := "VSEN ST6 HOLDFAST RH2 HP UP",
                           in_sensor_wp := "VSEN ST6 HOLDFAST RH2 WP DOWN",
                           in_ez_hp := "VALVE ST6 HOLDFAST RH2 HP UP",
                           in_ez_wp := "VALVE ST6 HOLDFAST RH2 WP DOWN",
                           in_ez_idle := "DBVALVES"."ST6 HOLDFAST RH2".test.IDLE_DUMMY,
                           out_in_hp => "DBVALVES"."ST6 HOLDFAST RH2".out.in_hp,
                           out_in_wp => "DBVALVES"."ST6 HOLDFAST RH2".out.in_wp,
                           out_idle => "DBVALVES"."ST6 HOLDFAST RH2".out.in_idle,
                           out_status => "DBVALVES"."ST6 HOLDFAST RH2".out.status);
END_REGION

REGION Network 165: [32] ST6 ROTATION LH
   RUNG wire#powerrail
      "INST ST6 ROTATION LH"(in_safety := wire#w1, in_move_hp := "DBVALVES"."ST6 ROTATION LH".in.move_hp, in_move_wp := "DBVALVES"."ST6 ROTATION LH".in.move_wp, in_move_idle := "DBVALVES"."ST6 ROTATION LH".in.move_idle, in_sensor_hp := "VSEN ST6 ROTATION LH HP LEFT", in_sensor_wp := "VSEN ST6 ROTATION LH WP RIGHT", in_ez_hp := "VALVE ST6 ROTATION LH HP LEFT", in_ez_wp := "VALVE ST6 ROTATION LH WP RIGHT", in_ez_idle := "DBVALVES"."ST6 ROTATION LH".test.IDLE_DUMMY, out_in_hp => "DBVALVES"."ST6 ROTATION LH".out.in_hp, out_in_wp => "DBVALVES"."ST6 ROTATION LH".out.in_wp, out_idle => "DBVALVES"."ST6 ROTATION LH".out.in_idle, out_status => "DBVALVES"."ST6 ROTATION LH".out.status)
   END_RUNG
   RUNG wire#powerrail
      Contact( "SIRIUS ESTOP" )
      Contact( "SIRIUS CURTAIN" )
   END_RUNG wire#w1
   // the same network as SCL:
   "INST ST6 ROTATION LH"(in_safety := "SIRIUS ESTOP" AND "SIRIUS CURTAIN",   // "3STATE_PISTON"
                          in_move_hp := "DBVALVES"."ST6 ROTATION LH".in.move_hp,
                          in_move_wp := "DBVALVES"."ST6 ROTATION LH".in.move_wp,
                          in_move_idle := "DBVALVES"."ST6 ROTATION LH".in.move_idle,
                          in_sensor_hp := "VSEN ST6 ROTATION LH HP LEFT",
                          in_sensor_wp := "VSEN ST6 ROTATION LH WP RIGHT",
                          in_ez_hp := "VALVE ST6 ROTATION LH HP LEFT",
                          in_ez_wp := "VALVE ST6 ROTATION LH WP RIGHT",
                          in_ez_idle := "DBVALVES"."ST6 ROTATION LH".test.IDLE_DUMMY,
                          out_in_hp => "DBVALVES"."ST6 ROTATION LH".out.in_hp,
                          out_in_wp => "DBVALVES"."ST6 ROTATION LH".out.in_wp,
                          out_idle => "DBVALVES"."ST6 ROTATION LH".out.in_idle,
                          out_status => "DBVALVES"."ST6 ROTATION LH".out.status);
END_REGION

REGION Network 166: [33] ST6 ROTATION RH
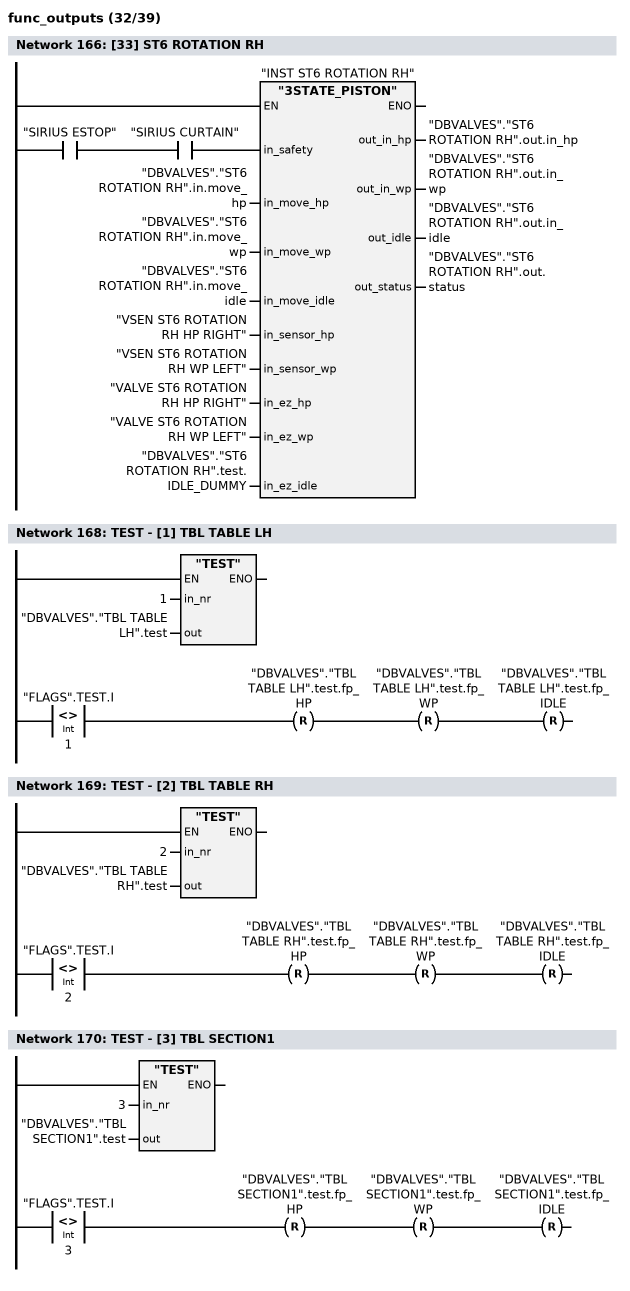
   RUNG wire#powerrail
      "INST ST6 ROTATION RH"(in_safety := wire#w1, in_move_hp := "DBVALVES"."ST6 ROTATION RH".in.move_hp, in_move_wp := "DBVALVES"."ST6 ROTATION RH".in.move_wp, in_move_idle := "DBVALVES"."ST6 ROTATION RH".in.move_idle, in_sensor_hp := "VSEN ST6 ROTATION RH HP RIGHT", in_sensor_wp := "VSEN ST6 ROTATION RH WP LEFT", in_ez_hp := "VALVE ST6 ROTATION RH HP RIGHT", in_ez_wp := "VALVE ST6 ROTATION RH WP LEFT", in_ez_idle := "DBVALVES"."ST6 ROTATION RH".test.IDLE_DUMMY, out_in_hp => "DBVALVES"."ST6 ROTATION RH".out.in_hp, out_in_wp => "DBVALVES"."ST6 ROTATION RH".out.in_wp, out_idle => "DBVALVES"."ST6 ROTATION RH".out.in_idle, out_status => "DBVALVES"."ST6 ROTATION RH".out.status)
   END_RUNG
   RUNG wire#powerrail
      Contact( "SIRIUS ESTOP" )
      Contact( "SIRIUS CURTAIN" )
   END_RUNG wire#w1
   // the same network as SCL:
   "INST ST6 ROTATION RH"(in_safety := "SIRIUS ESTOP" AND "SIRIUS CURTAIN",   // "3STATE_PISTON"
                          in_move_hp := "DBVALVES"."ST6 ROTATION RH".in.move_hp,
                          in_move_wp := "DBVALVES"."ST6 ROTATION RH".in.move_wp,
                          in_move_idle := "DBVALVES"."ST6 ROTATION RH".in.move_idle,
                          in_sensor_hp := "VSEN ST6 ROTATION RH HP RIGHT",
                          in_sensor_wp := "VSEN ST6 ROTATION RH WP LEFT",
                          in_ez_hp := "VALVE ST6 ROTATION RH HP RIGHT",
                          in_ez_wp := "VALVE ST6 ROTATION RH WP LEFT",
                          in_ez_idle := "DBVALVES"."ST6 ROTATION RH".test.IDLE_DUMMY,
                          out_in_hp => "DBVALVES"."ST6 ROTATION RH".out.in_hp,
                          out_in_wp => "DBVALVES"."ST6 ROTATION RH".out.in_wp,
                          out_idle => "DBVALVES"."ST6 ROTATION RH".out.in_idle,
                          out_status => "DBVALVES"."ST6 ROTATION RH".out.status);
END_REGION

REGION Network 167: ======= TESTS =======
END_REGION

REGION Network 168: TEST - [1] TBL TABLE LH
   RUNG wire#powerrail
      "TEST"(in_nr := 1, out := "DBVALVES"."TBL TABLE LH".test)
   END_RUNG
   RUNG wire#powerrail
      { S7_Templates := "SrcType := Int" } NE_Contact(in1 := "FLAGS".TEST.I, in2 := 1)
      R_Coil( "DBVALVES"."TBL TABLE LH".test.fp_HP )
      R_Coil( "DBVALVES"."TBL TABLE LH".test.fp_WP )
      R_Coil( "DBVALVES"."TBL TABLE LH".test.fp_IDLE )
   END_RUNG
   // the same network as SCL:
   "TEST"(in_nr := 1, out := "DBVALVES"."TBL TABLE LH".test);
   IF "FLAGS".TEST.I <> 1 THEN
       "DBVALVES"."TBL TABLE LH".test.fp_HP := FALSE;
       "DBVALVES"."TBL TABLE LH".test.fp_WP := FALSE;
       "DBVALVES"."TBL TABLE LH".test.fp_IDLE := FALSE;
   END_IF;
END_REGION

REGION Network 169: TEST - [2] TBL TABLE RH
   RUNG wire#powerrail
      "TEST"(in_nr := 2, out := "DBVALVES"."TBL TABLE RH".test)
   END_RUNG
   RUNG wire#powerrail
      { S7_Templates := "SrcType := Int" } NE_Contact(in1 := "FLAGS".TEST.I, in2 := 2)
      R_Coil( "DBVALVES"."TBL TABLE RH".test.fp_HP )
      R_Coil( "DBVALVES"."TBL TABLE RH".test.fp_WP )
      R_Coil( "DBVALVES"."TBL TABLE RH".test.fp_IDLE )
   END_RUNG
   // the same network as SCL:
   "TEST"(in_nr := 2, out := "DBVALVES"."TBL TABLE RH".test);
   IF "FLAGS".TEST.I <> 2 THEN
       "DBVALVES"."TBL TABLE RH".test.fp_HP := FALSE;
       "DBVALVES"."TBL TABLE RH".test.fp_WP := FALSE;
       "DBVALVES"."TBL TABLE RH".test.fp_IDLE := FALSE;
   END_IF;
END_REGION

REGION Network 170: TEST - [3] TBL SECTION1
   RUNG wire#powerrail
      "TEST"(in_nr := 3, out := "DBVALVES"."TBL SECTION1".test)
   END_RUNG
   RUNG wire#powerrail
      { S7_Templates := "SrcType := Int" } NE_Contact(in1 := "FLAGS".TEST.I, in2 := 3)
      R_Coil( "DBVALVES"."TBL SECTION1".test.fp_HP )
      R_Coil( "DBVALVES"."TBL SECTION1".test.fp_WP )
      R_Coil( "DBVALVES"."TBL SECTION1".test.fp_IDLE )
   END_RUNG
   // the same network as SCL:
   "TEST"(in_nr := 3, out := "DBVALVES"."TBL SECTION1".test);
   IF "FLAGS".TEST.I <> 3 THEN
       "DBVALVES"."TBL SECTION1".test.fp_HP := FALSE;
       "DBVALVES"."TBL SECTION1".test.fp_WP := FALSE;
       "DBVALVES"."TBL SECTION1".test.fp_IDLE := FALSE;
   END_IF;
END_REGION

REGION Network 171: TEST - [4] TBL SECTION2
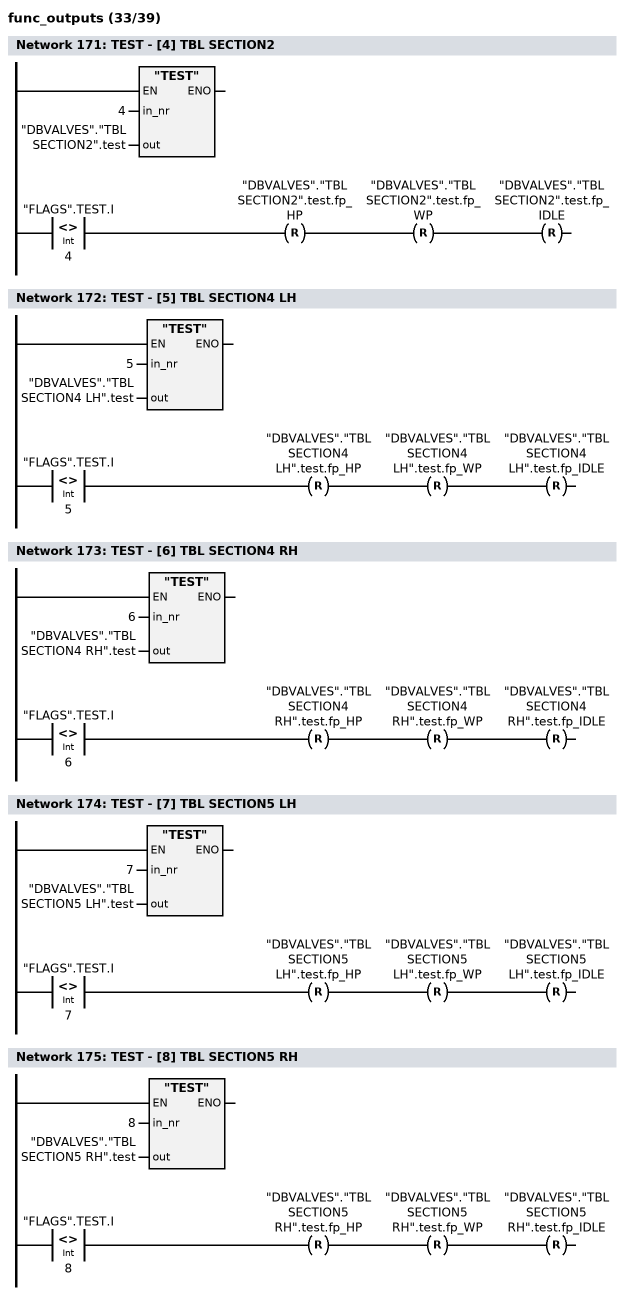
   RUNG wire#powerrail
      "TEST"(in_nr := 4, out := "DBVALVES"."TBL SECTION2".test)
   END_RUNG
   RUNG wire#powerrail
      { S7_Templates := "SrcType := Int" } NE_Contact(in1 := "FLAGS".TEST.I, in2 := 4)
      R_Coil( "DBVALVES"."TBL SECTION2".test.fp_HP )
      R_Coil( "DBVALVES"."TBL SECTION2".test.fp_WP )
      R_Coil( "DBVALVES"."TBL SECTION2".test.fp_IDLE )
   END_RUNG
   // the same network as SCL:
   "TEST"(in_nr := 4, out := "DBVALVES"."TBL SECTION2".test);
   IF "FLAGS".TEST.I <> 4 THEN
       "DBVALVES"."TBL SECTION2".test.fp_HP := FALSE;
       "DBVALVES"."TBL SECTION2".test.fp_WP := FALSE;
       "DBVALVES"."TBL SECTION2".test.fp_IDLE := FALSE;
   END_IF;
END_REGION

REGION Network 172: TEST - [5] TBL SECTION4 LH
   RUNG wire#powerrail
      "TEST"(in_nr := 5, out := "DBVALVES"."TBL SECTION4 LH".test)
   END_RUNG
   RUNG wire#powerrail
      { S7_Templates := "SrcType := Int" } NE_Contact(in1 := "FLAGS".TEST.I, in2 := 5)
      R_Coil( "DBVALVES"."TBL SECTION4 LH".test.fp_HP )
      R_Coil( "DBVALVES"."TBL SECTION4 LH".test.fp_WP )
      R_Coil( "DBVALVES"."TBL SECTION4 LH".test.fp_IDLE )
   END_RUNG
   // the same network as SCL:
   "TEST"(in_nr := 5, out := "DBVALVES"."TBL SECTION4 LH".test);
   IF "FLAGS".TEST.I <> 5 THEN
       "DBVALVES"."TBL SECTION4 LH".test.fp_HP := FALSE;
       "DBVALVES"."TBL SECTION4 LH".test.fp_WP := FALSE;
       "DBVALVES"."TBL SECTION4 LH".test.fp_IDLE := FALSE;
   END_IF;
END_REGION

REGION Network 173: TEST - [6] TBL SECTION4 RH
   RUNG wire#powerrail
      "TEST"(in_nr := 6, out := "DBVALVES"."TBL SECTION4 RH".test)
   END_RUNG
   RUNG wire#powerrail
      { S7_Templates := "SrcType := Int" } NE_Contact(in1 := "FLAGS".TEST.I, in2 := 6)
      R_Coil( "DBVALVES"."TBL SECTION4 RH".test.fp_HP )
      R_Coil( "DBVALVES"."TBL SECTION4 RH".test.fp_WP )
      R_Coil( "DBVALVES"."TBL SECTION4 RH".test.fp_IDLE )
   END_RUNG
   // the same network as SCL:
   "TEST"(in_nr := 6, out := "DBVALVES"."TBL SECTION4 RH".test);
   IF "FLAGS".TEST.I <> 6 THEN
       "DBVALVES"."TBL SECTION4 RH".test.fp_HP := FALSE;
       "DBVALVES"."TBL SECTION4 RH".test.fp_WP := FALSE;
       "DBVALVES"."TBL SECTION4 RH".test.fp_IDLE := FALSE;
   END_IF;
END_REGION

REGION Network 174: TEST - [7] TBL SECTION5 LH
   RUNG wire#powerrail
      "TEST"(in_nr := 7, out := "DBVALVES"."TBL SECTION5 LH".test)
   END_RUNG
   RUNG wire#powerrail
      { S7_Templates := "SrcType := Int" } NE_Contact(in1 := "FLAGS".TEST.I, in2 := 7)
      R_Coil( "DBVALVES"."TBL SECTION5 LH".test.fp_HP )
      R_Coil( "DBVALVES"."TBL SECTION5 LH".test.fp_WP )
      R_Coil( "DBVALVES"."TBL SECTION5 LH".test.fp_IDLE )
   END_RUNG
   // the same network as SCL:
   "TEST"(in_nr := 7, out := "DBVALVES"."TBL SECTION5 LH".test);
   IF "FLAGS".TEST.I <> 7 THEN
       "DBVALVES"."TBL SECTION5 LH".test.fp_HP := FALSE;
       "DBVALVES"."TBL SECTION5 LH".test.fp_WP := FALSE;
       "DBVALVES"."TBL SECTION5 LH".test.fp_IDLE := FALSE;
   END_IF;
END_REGION

REGION Network 175: TEST - [8] TBL SECTION5 RH
   RUNG wire#powerrail
      "TEST"(in_nr := 8, out := "DBVALVES"."TBL SECTION5 RH".test)
   END_RUNG
   RUNG wire#powerrail
      { S7_Templates := "SrcType := Int" } NE_Contact(in1 := "FLAGS".TEST.I, in2 := 8)
      R_Coil( "DBVALVES"."TBL SECTION5 RH".test.fp_HP )
      R_Coil( "DBVALVES"."TBL SECTION5 RH".test.fp_WP )
      R_Coil( "DBVALVES"."TBL SECTION5 RH".test.fp_IDLE )
   END_RUNG
   // the same network as SCL:
   "TEST"(in_nr := 8, out := "DBVALVES"."TBL SECTION5 RH".test);
   IF "FLAGS".TEST.I <> 8 THEN
       "DBVALVES"."TBL SECTION5 RH".test.fp_HP := FALSE;
       "DBVALVES"."TBL SECTION5 RH".test.fp_WP := FALSE;
       "DBVALVES"."TBL SECTION5 RH".test.fp_IDLE := FALSE;
   END_IF;
END_REGION

REGION Network 176: TEST - [9] TBL POSITIONING LH
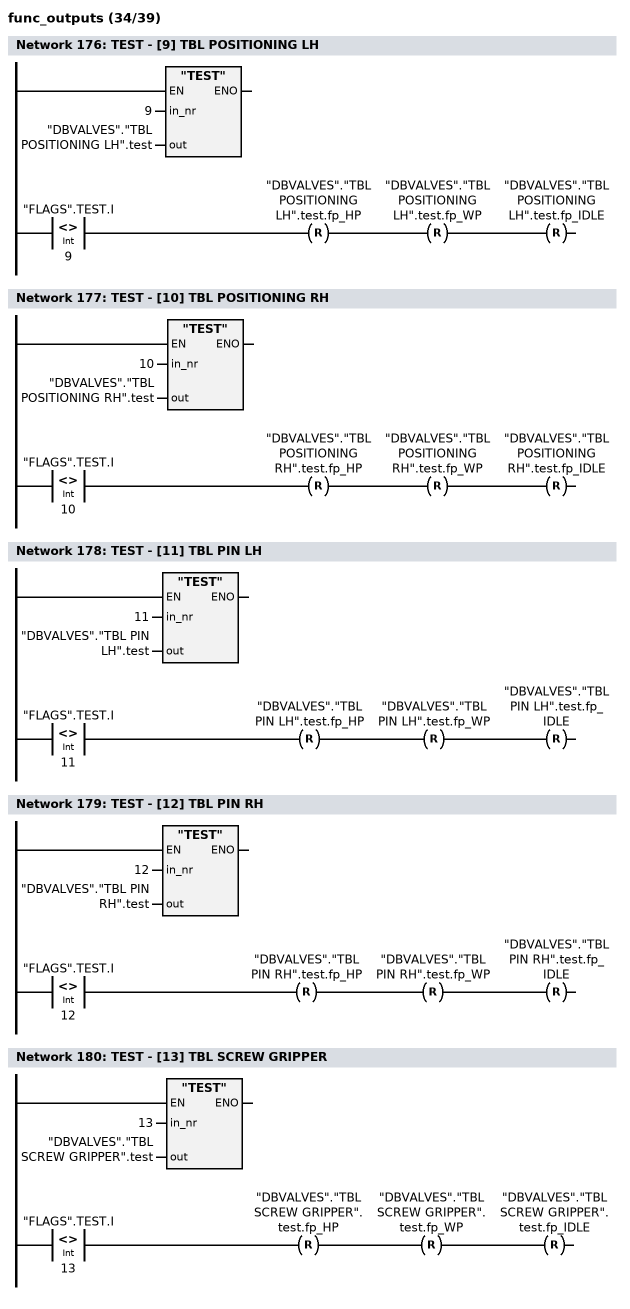
   RUNG wire#powerrail
      "TEST"(in_nr := 9, out := "DBVALVES"."TBL POSITIONING LH".test)
   END_RUNG
   RUNG wire#powerrail
      { S7_Templates := "SrcType := Int" } NE_Contact(in1 := "FLAGS".TEST.I, in2 := 9)
      R_Coil( "DBVALVES"."TBL POSITIONING LH".test.fp_HP )
      R_Coil( "DBVALVES"."TBL POSITIONING LH".test.fp_WP )
      R_Coil( "DBVALVES"."TBL POSITIONING LH".test.fp_IDLE )
   END_RUNG
   // the same network as SCL:
   "TEST"(in_nr := 9, out := "DBVALVES"."TBL POSITIONING LH".test);
   IF "FLAGS".TEST.I <> 9 THEN
       "DBVALVES"."TBL POSITIONING LH".test.fp_HP := FALSE;
       "DBVALVES"."TBL POSITIONING LH".test.fp_WP := FALSE;
       "DBVALVES"."TBL POSITIONING LH".test.fp_IDLE := FALSE;
   END_IF;
END_REGION

REGION Network 177: TEST - [10] TBL POSITIONING RH
   RUNG wire#powerrail
      "TEST"(in_nr := 10, out := "DBVALVES"."TBL POSITIONING RH".test)
   END_RUNG
   RUNG wire#powerrail
      { S7_Templates := "SrcType := Int" } NE_Contact(in1 := "FLAGS".TEST.I, in2 := 10)
      R_Coil( "DBVALVES"."TBL POSITIONING RH".test.fp_HP )
      R_Coil( "DBVALVES"."TBL POSITIONING RH".test.fp_WP )
      R_Coil( "DBVALVES"."TBL POSITIONING RH".test.fp_IDLE )
   END_RUNG
   // the same network as SCL:
   "TEST"(in_nr := 10, out := "DBVALVES"."TBL POSITIONING RH".test);
   IF "FLAGS".TEST.I <> 10 THEN
       "DBVALVES"."TBL POSITIONING RH".test.fp_HP := FALSE;
       "DBVALVES"."TBL POSITIONING RH".test.fp_WP := FALSE;
       "DBVALVES"."TBL POSITIONING RH".test.fp_IDLE := FALSE;
   END_IF;
END_REGION

REGION Network 178: TEST - [11] TBL PIN LH
   RUNG wire#powerrail
      "TEST"(in_nr := 11, out := "DBVALVES"."TBL PIN LH".test)
   END_RUNG
   RUNG wire#powerrail
      { S7_Templates := "SrcType := Int" } NE_Contact(in1 := "FLAGS".TEST.I, in2 := 11)
      R_Coil( "DBVALVES"."TBL PIN LH".test.fp_HP )
      R_Coil( "DBVALVES"."TBL PIN LH".test.fp_WP )
      R_Coil( "DBVALVES"."TBL PIN LH".test.fp_IDLE )
   END_RUNG
   // the same network as SCL:
   "TEST"(in_nr := 11, out := "DBVALVES"."TBL PIN LH".test);
   IF "FLAGS".TEST.I <> 11 THEN
       "DBVALVES"."TBL PIN LH".test.fp_HP := FALSE;
       "DBVALVES"."TBL PIN LH".test.fp_WP := FALSE;
       "DBVALVES"."TBL PIN LH".test.fp_IDLE := FALSE;
   END_IF;
END_REGION

REGION Network 179: TEST - [12] TBL PIN RH
   RUNG wire#powerrail
      "TEST"(in_nr := 12, out := "DBVALVES"."TBL PIN RH".test)
   END_RUNG
   RUNG wire#powerrail
      { S7_Templates := "SrcType := Int" } NE_Contact(in1 := "FLAGS".TEST.I, in2 := 12)
      R_Coil( "DBVALVES"."TBL PIN RH".test.fp_HP )
      R_Coil( "DBVALVES"."TBL PIN RH".test.fp_WP )
      R_Coil( "DBVALVES"."TBL PIN RH".test.fp_IDLE )
   END_RUNG
   // the same network as SCL:
   "TEST"(in_nr := 12, out := "DBVALVES"."TBL PIN RH".test);
   IF "FLAGS".TEST.I <> 12 THEN
       "DBVALVES"."TBL PIN RH".test.fp_HP := FALSE;
       "DBVALVES"."TBL PIN RH".test.fp_WP := FALSE;
       "DBVALVES"."TBL PIN RH".test.fp_IDLE := FALSE;
   END_IF;
END_REGION

REGION Network 180: TEST - [13] TBL SCREW GRIPPER
   RUNG wire#powerrail
      "TEST"(in_nr := 13, out := "DBVALVES"."TBL SCREW GRIPPER".test)
   END_RUNG
   RUNG wire#powerrail
      { S7_Templates := "SrcType := Int" } NE_Contact(in1 := "FLAGS".TEST.I, in2 := 13)
      R_Coil( "DBVALVES"."TBL SCREW GRIPPER".test.fp_HP )
      R_Coil( "DBVALVES"."TBL SCREW GRIPPER".test.fp_WP )
      R_Coil( "DBVALVES"."TBL SCREW GRIPPER".test.fp_IDLE )
   END_RUNG
   // the same network as SCL:
   "TEST"(in_nr := 13, out := "DBVALVES"."TBL SCREW GRIPPER".test);
   IF "FLAGS".TEST.I <> 13 THEN
       "DBVALVES"."TBL SCREW GRIPPER".test.fp_HP := FALSE;
       "DBVALVES"."TBL SCREW GRIPPER".test.fp_WP := FALSE;
       "DBVALVES"."TBL SCREW GRIPPER".test.fp_IDLE := FALSE;
   END_IF;
END_REGION

REGION Network 181: TEST - [14] TBL WRAP GRIPPER
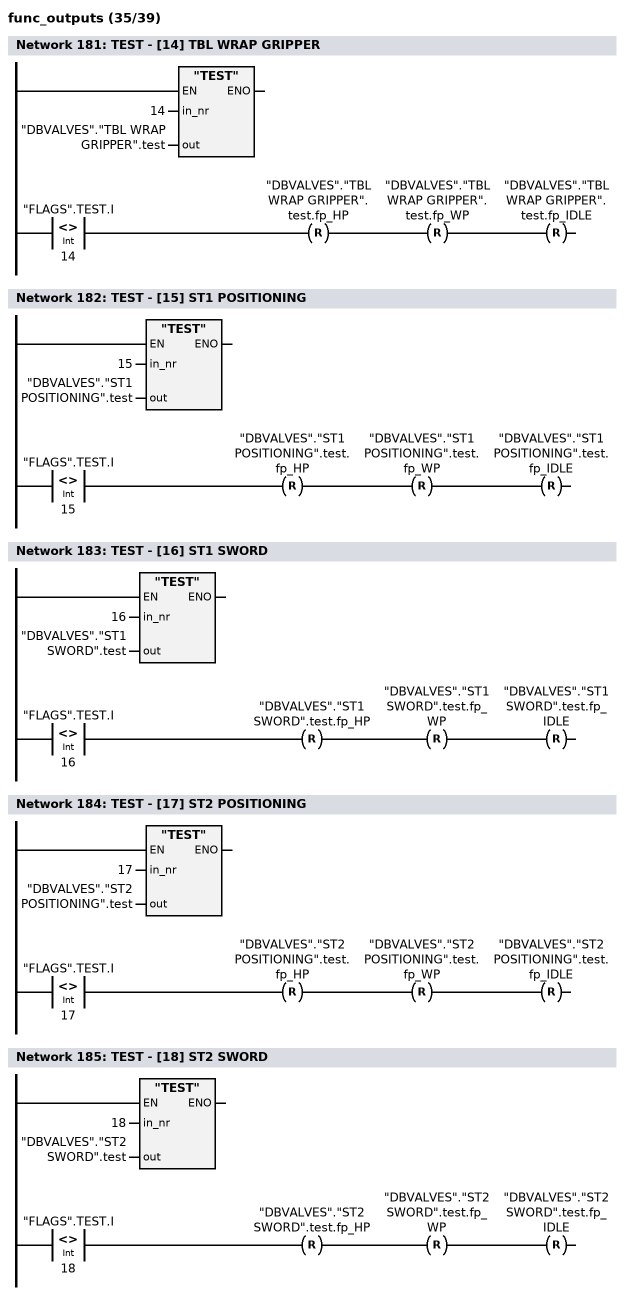
   RUNG wire#powerrail
      "TEST"(in_nr := 14, out := "DBVALVES"."TBL WRAP GRIPPER".test)
   END_RUNG
   RUNG wire#powerrail
      { S7_Templates := "SrcType := Int" } NE_Contact(in1 := "FLAGS".TEST.I, in2 := 14)
      R_Coil( "DBVALVES"."TBL WRAP GRIPPER".test.fp_HP )
      R_Coil( "DBVALVES"."TBL WRAP GRIPPER".test.fp_WP )
      R_Coil( "DBVALVES"."TBL WRAP GRIPPER".test.fp_IDLE )
   END_RUNG
   // the same network as SCL:
   "TEST"(in_nr := 14, out := "DBVALVES"."TBL WRAP GRIPPER".test);
   IF "FLAGS".TEST.I <> 14 THEN
       "DBVALVES"."TBL WRAP GRIPPER".test.fp_HP := FALSE;
       "DBVALVES"."TBL WRAP GRIPPER".test.fp_WP := FALSE;
       "DBVALVES"."TBL WRAP GRIPPER".test.fp_IDLE := FALSE;
   END_IF;
END_REGION

REGION Network 182: TEST - [15] ST1 POSITIONING
   RUNG wire#powerrail
      "TEST"(in_nr := 15, out := "DBVALVES"."ST1 POSITIONING".test)
   END_RUNG
   RUNG wire#powerrail
      { S7_Templates := "SrcType := Int" } NE_Contact(in1 := "FLAGS".TEST.I, in2 := 15)
      R_Coil( "DBVALVES"."ST1 POSITIONING".test.fp_HP )
      R_Coil( "DBVALVES"."ST1 POSITIONING".test.fp_WP )
      R_Coil( "DBVALVES"."ST1 POSITIONING".test.fp_IDLE )
   END_RUNG
   // the same network as SCL:
   "TEST"(in_nr := 15, out := "DBVALVES"."ST1 POSITIONING".test);
   IF "FLAGS".TEST.I <> 15 THEN
       "DBVALVES"."ST1 POSITIONING".test.fp_HP := FALSE;
       "DBVALVES"."ST1 POSITIONING".test.fp_WP := FALSE;
       "DBVALVES"."ST1 POSITIONING".test.fp_IDLE := FALSE;
   END_IF;
END_REGION

REGION Network 183: TEST - [16] ST1 SWORD
   RUNG wire#powerrail
      "TEST"(in_nr := 16, out := "DBVALVES"."ST1 SWORD".test)
   END_RUNG
   RUNG wire#powerrail
      { S7_Templates := "SrcType := Int" } NE_Contact(in1 := "FLAGS".TEST.I, in2 := 16)
      R_Coil( "DBVALVES"."ST1 SWORD".test.fp_HP )
      R_Coil( "DBVALVES"."ST1 SWORD".test.fp_WP )
      R_Coil( "DBVALVES"."ST1 SWORD".test.fp_IDLE )
   END_RUNG
   // the same network as SCL:
   "TEST"(in_nr := 16, out := "DBVALVES"."ST1 SWORD".test);
   IF "FLAGS".TEST.I <> 16 THEN
       "DBVALVES"."ST1 SWORD".test.fp_HP := FALSE;
       "DBVALVES"."ST1 SWORD".test.fp_WP := FALSE;
       "DBVALVES"."ST1 SWORD".test.fp_IDLE := FALSE;
   END_IF;
END_REGION

REGION Network 184: TEST - [17] ST2 POSITIONING
   RUNG wire#powerrail
      "TEST"(in_nr := 17, out := "DBVALVES"."ST2 POSITIONING".test)
   END_RUNG
   RUNG wire#powerrail
      { S7_Templates := "SrcType := Int" } NE_Contact(in1 := "FLAGS".TEST.I, in2 := 17)
      R_Coil( "DBVALVES"."ST2 POSITIONING".test.fp_HP )
      R_Coil( "DBVALVES"."ST2 POSITIONING".test.fp_WP )
      R_Coil( "DBVALVES"."ST2 POSITIONING".test.fp_IDLE )
   END_RUNG
   // the same network as SCL:
   "TEST"(in_nr := 17, out := "DBVALVES"."ST2 POSITIONING".test);
   IF "FLAGS".TEST.I <> 17 THEN
       "DBVALVES"."ST2 POSITIONING".test.fp_HP := FALSE;
       "DBVALVES"."ST2 POSITIONING".test.fp_WP := FALSE;
       "DBVALVES"."ST2 POSITIONING".test.fp_IDLE := FALSE;
   END_IF;
END_REGION

REGION Network 185: TEST - [18] ST2 SWORD
   RUNG wire#powerrail
      "TEST"(in_nr := 18, out := "DBVALVES"."ST2 SWORD".test)
   END_RUNG
   RUNG wire#powerrail
      { S7_Templates := "SrcType := Int" } NE_Contact(in1 := "FLAGS".TEST.I, in2 := 18)
      R_Coil( "DBVALVES"."ST2 SWORD".test.fp_HP )
      R_Coil( "DBVALVES"."ST2 SWORD".test.fp_WP )
      R_Coil( "DBVALVES"."ST2 SWORD".test.fp_IDLE )
   END_RUNG
   // the same network as SCL:
   "TEST"(in_nr := 18, out := "DBVALVES"."ST2 SWORD".test);
   IF "FLAGS".TEST.I <> 18 THEN
       "DBVALVES"."ST2 SWORD".test.fp_HP := FALSE;
       "DBVALVES"."ST2 SWORD".test.fp_WP := FALSE;
       "DBVALVES"."ST2 SWORD".test.fp_IDLE := FALSE;
   END_IF;
END_REGION

REGION Network 186: TEST - [19] ST3 POSITIONING
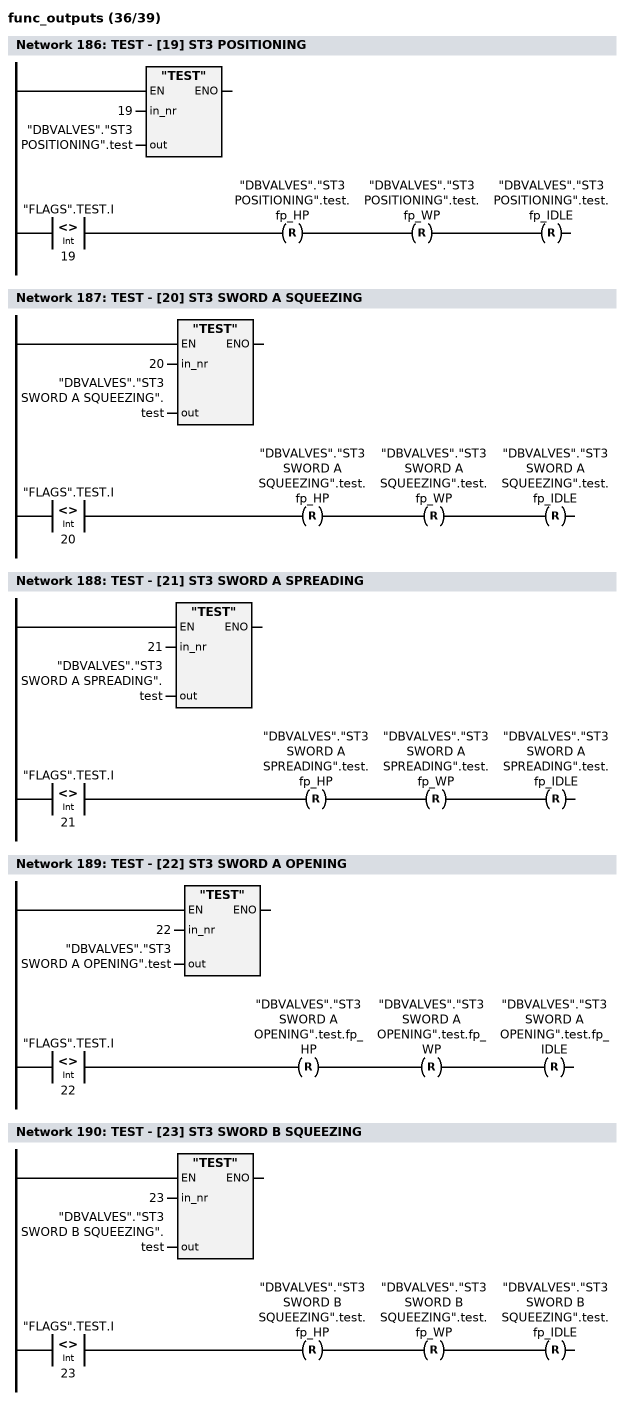
   RUNG wire#powerrail
      "TEST"(in_nr := 19, out := "DBVALVES"."ST3 POSITIONING".test)
   END_RUNG
   RUNG wire#powerrail
      { S7_Templates := "SrcType := Int" } NE_Contact(in1 := "FLAGS".TEST.I, in2 := 19)
      R_Coil( "DBVALVES"."ST3 POSITIONING".test.fp_HP )
      R_Coil( "DBVALVES"."ST3 POSITIONING".test.fp_WP )
      R_Coil( "DBVALVES"."ST3 POSITIONING".test.fp_IDLE )
   END_RUNG
   // the same network as SCL:
   "TEST"(in_nr := 19, out := "DBVALVES"."ST3 POSITIONING".test);
   IF "FLAGS".TEST.I <> 19 THEN
       "DBVALVES"."ST3 POSITIONING".test.fp_HP := FALSE;
       "DBVALVES"."ST3 POSITIONING".test.fp_WP := FALSE;
       "DBVALVES"."ST3 POSITIONING".test.fp_IDLE := FALSE;
   END_IF;
END_REGION

REGION Network 187: TEST - [20] ST3 SWORD A SQUEEZING
   RUNG wire#powerrail
      "TEST"(in_nr := 20, out := "DBVALVES"."ST3 SWORD A SQUEEZING".test)
   END_RUNG
   RUNG wire#powerrail
      { S7_Templates := "SrcType := Int" } NE_Contact(in1 := "FLAGS".TEST.I, in2 := 20)
      R_Coil( "DBVALVES"."ST3 SWORD A SQUEEZING".test.fp_HP )
      R_Coil( "DBVALVES"."ST3 SWORD A SQUEEZING".test.fp_WP )
      R_Coil( "DBVALVES"."ST3 SWORD A SQUEEZING".test.fp_IDLE )
   END_RUNG
   // the same network as SCL:
   "TEST"(in_nr := 20, out := "DBVALVES"."ST3 SWORD A SQUEEZING".test);
   IF "FLAGS".TEST.I <> 20 THEN
       "DBVALVES"."ST3 SWORD A SQUEEZING".test.fp_HP := FALSE;
       "DBVALVES"."ST3 SWORD A SQUEEZING".test.fp_WP := FALSE;
       "DBVALVES"."ST3 SWORD A SQUEEZING".test.fp_IDLE := FALSE;
   END_IF;
END_REGION

REGION Network 188: TEST - [21] ST3 SWORD A SPREADING
   RUNG wire#powerrail
      "TEST"(in_nr := 21, out := "DBVALVES"."ST3 SWORD A SPREADING".test)
   END_RUNG
   RUNG wire#powerrail
      { S7_Templates := "SrcType := Int" } NE_Contact(in1 := "FLAGS".TEST.I, in2 := 21)
      R_Coil( "DBVALVES"."ST3 SWORD A SPREADING".test.fp_HP )
      R_Coil( "DBVALVES"."ST3 SWORD A SPREADING".test.fp_WP )
      R_Coil( "DBVALVES"."ST3 SWORD A SPREADING".test.fp_IDLE )
   END_RUNG
   // the same network as SCL:
   "TEST"(in_nr := 21, out := "DBVALVES"."ST3 SWORD A SPREADING".test);
   IF "FLAGS".TEST.I <> 21 THEN
       "DBVALVES"."ST3 SWORD A SPREADING".test.fp_HP := FALSE;
       "DBVALVES"."ST3 SWORD A SPREADING".test.fp_WP := FALSE;
       "DBVALVES"."ST3 SWORD A SPREADING".test.fp_IDLE := FALSE;
   END_IF;
END_REGION

REGION Network 189: TEST - [22] ST3 SWORD A OPENING
   RUNG wire#powerrail
      "TEST"(in_nr := 22, out := "DBVALVES"."ST3 SWORD A OPENING".test)
   END_RUNG
   RUNG wire#powerrail
      { S7_Templates := "SrcType := Int" } NE_Contact(in1 := "FLAGS".TEST.I, in2 := 22)
      R_Coil( "DBVALVES"."ST3 SWORD A OPENING".test.fp_HP )
      R_Coil( "DBVALVES"."ST3 SWORD A OPENING".test.fp_WP )
      R_Coil( "DBVALVES"."ST3 SWORD A OPENING".test.fp_IDLE )
   END_RUNG
   // the same network as SCL:
   "TEST"(in_nr := 22, out := "DBVALVES"."ST3 SWORD A OPENING".test);
   IF "FLAGS".TEST.I <> 22 THEN
       "DBVALVES"."ST3 SWORD A OPENING".test.fp_HP := FALSE;
       "DBVALVES"."ST3 SWORD A OPENING".test.fp_WP := FALSE;
       "DBVALVES"."ST3 SWORD A OPENING".test.fp_IDLE := FALSE;
   END_IF;
END_REGION

REGION Network 190: TEST - [23] ST3 SWORD B SQUEEZING
   RUNG wire#powerrail
      "TEST"(in_nr := 23, out := "DBVALVES"."ST3 SWORD B SQUEEZING".test)
   END_RUNG
   RUNG wire#powerrail
      { S7_Templates := "SrcType := Int" } NE_Contact(in1 := "FLAGS".TEST.I, in2 := 23)
      R_Coil( "DBVALVES"."ST3 SWORD B SQUEEZING".test.fp_HP )
      R_Coil( "DBVALVES"."ST3 SWORD B SQUEEZING".test.fp_WP )
      R_Coil( "DBVALVES"."ST3 SWORD B SQUEEZING".test.fp_IDLE )
   END_RUNG
   // the same network as SCL:
   "TEST"(in_nr := 23, out := "DBVALVES"."ST3 SWORD B SQUEEZING".test);
   IF "FLAGS".TEST.I <> 23 THEN
       "DBVALVES"."ST3 SWORD B SQUEEZING".test.fp_HP := FALSE;
       "DBVALVES"."ST3 SWORD B SQUEEZING".test.fp_WP := FALSE;
       "DBVALVES"."ST3 SWORD B SQUEEZING".test.fp_IDLE := FALSE;
   END_IF;
END_REGION

REGION Network 191: TEST - [24] ST3 SWORD B SPREADING
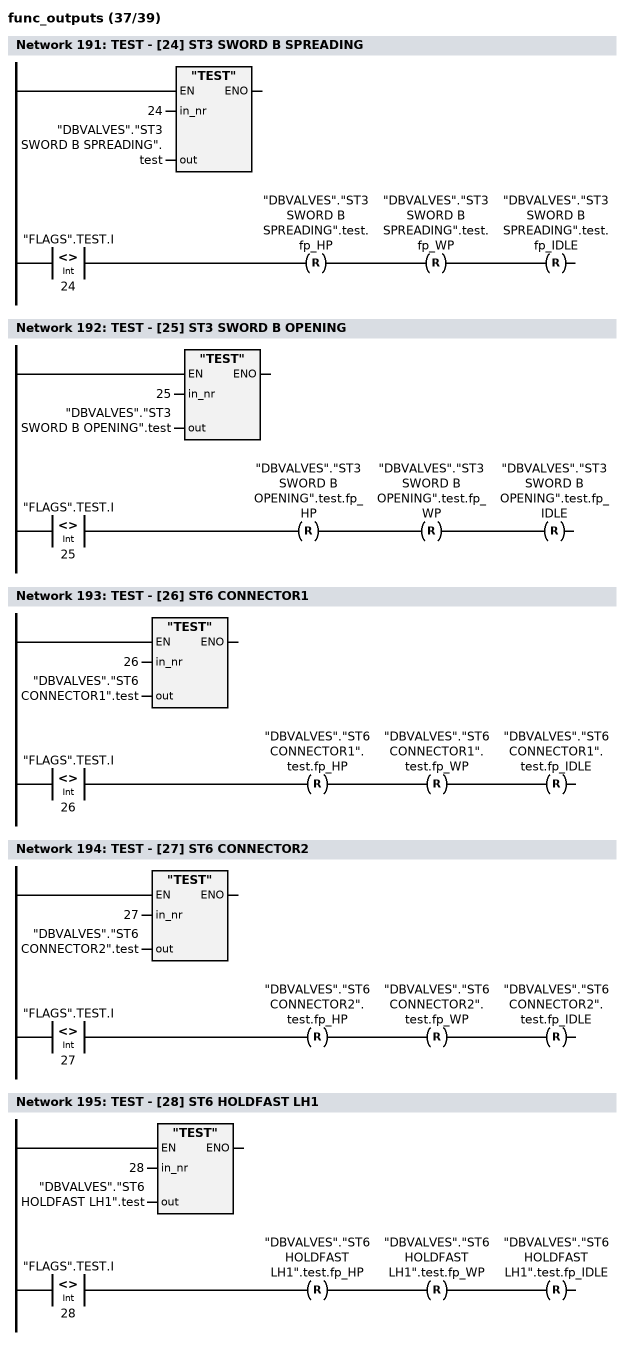
   RUNG wire#powerrail
      "TEST"(in_nr := 24, out := "DBVALVES"."ST3 SWORD B SPREADING".test)
   END_RUNG
   RUNG wire#powerrail
      { S7_Templates := "SrcType := Int" } NE_Contact(in1 := "FLAGS".TEST.I, in2 := 24)
      R_Coil( "DBVALVES"."ST3 SWORD B SPREADING".test.fp_HP )
      R_Coil( "DBVALVES"."ST3 SWORD B SPREADING".test.fp_WP )
      R_Coil( "DBVALVES"."ST3 SWORD B SPREADING".test.fp_IDLE )
   END_RUNG
   // the same network as SCL:
   "TEST"(in_nr := 24, out := "DBVALVES"."ST3 SWORD B SPREADING".test);
   IF "FLAGS".TEST.I <> 24 THEN
       "DBVALVES"."ST3 SWORD B SPREADING".test.fp_HP := FALSE;
       "DBVALVES"."ST3 SWORD B SPREADING".test.fp_WP := FALSE;
       "DBVALVES"."ST3 SWORD B SPREADING".test.fp_IDLE := FALSE;
   END_IF;
END_REGION

REGION Network 192: TEST - [25] ST3 SWORD B OPENING
   RUNG wire#powerrail
      "TEST"(in_nr := 25, out := "DBVALVES"."ST3 SWORD B OPENING".test)
   END_RUNG
   RUNG wire#powerrail
      { S7_Templates := "SrcType := Int" } NE_Contact(in1 := "FLAGS".TEST.I, in2 := 25)
      R_Coil( "DBVALVES"."ST3 SWORD B OPENING".test.fp_HP )
      R_Coil( "DBVALVES"."ST3 SWORD B OPENING".test.fp_WP )
      R_Coil( "DBVALVES"."ST3 SWORD B OPENING".test.fp_IDLE )
   END_RUNG
   // the same network as SCL:
   "TEST"(in_nr := 25, out := "DBVALVES"."ST3 SWORD B OPENING".test);
   IF "FLAGS".TEST.I <> 25 THEN
       "DBVALVES"."ST3 SWORD B OPENING".test.fp_HP := FALSE;
       "DBVALVES"."ST3 SWORD B OPENING".test.fp_WP := FALSE;
       "DBVALVES"."ST3 SWORD B OPENING".test.fp_IDLE := FALSE;
   END_IF;
END_REGION

REGION Network 193: TEST - [26] ST6 CONNECTOR1
   RUNG wire#powerrail
      "TEST"(in_nr := 26, out := "DBVALVES"."ST6 CONNECTOR1".test)
   END_RUNG
   RUNG wire#powerrail
      { S7_Templates := "SrcType := Int" } NE_Contact(in1 := "FLAGS".TEST.I, in2 := 26)
      R_Coil( "DBVALVES"."ST6 CONNECTOR1".test.fp_HP )
      R_Coil( "DBVALVES"."ST6 CONNECTOR1".test.fp_WP )
      R_Coil( "DBVALVES"."ST6 CONNECTOR1".test.fp_IDLE )
   END_RUNG
   // the same network as SCL:
   "TEST"(in_nr := 26, out := "DBVALVES"."ST6 CONNECTOR1".test);
   IF "FLAGS".TEST.I <> 26 THEN
       "DBVALVES"."ST6 CONNECTOR1".test.fp_HP := FALSE;
       "DBVALVES"."ST6 CONNECTOR1".test.fp_WP := FALSE;
       "DBVALVES"."ST6 CONNECTOR1".test.fp_IDLE := FALSE;
   END_IF;
END_REGION

REGION Network 194: TEST - [27] ST6 CONNECTOR2
   RUNG wire#powerrail
      "TEST"(in_nr := 27, out := "DBVALVES"."ST6 CONNECTOR2".test)
   END_RUNG
   RUNG wire#powerrail
      { S7_Templates := "SrcType := Int" } NE_Contact(in1 := "FLAGS".TEST.I, in2 := 27)
      R_Coil( "DBVALVES"."ST6 CONNECTOR2".test.fp_HP )
      R_Coil( "DBVALVES"."ST6 CONNECTOR2".test.fp_WP )
      R_Coil( "DBVALVES"."ST6 CONNECTOR2".test.fp_IDLE )
   END_RUNG
   // the same network as SCL:
   "TEST"(in_nr := 27, out := "DBVALVES"."ST6 CONNECTOR2".test);
   IF "FLAGS".TEST.I <> 27 THEN
       "DBVALVES"."ST6 CONNECTOR2".test.fp_HP := FALSE;
       "DBVALVES"."ST6 CONNECTOR2".test.fp_WP := FALSE;
       "DBVALVES"."ST6 CONNECTOR2".test.fp_IDLE := FALSE;
   END_IF;
END_REGION

REGION Network 195: TEST - [28] ST6 HOLDFAST LH1
   RUNG wire#powerrail
      "TEST"(in_nr := 28, out := "DBVALVES"."ST6 HOLDFAST LH1".test)
   END_RUNG
   RUNG wire#powerrail
      { S7_Templates := "SrcType := Int" } NE_Contact(in1 := "FLAGS".TEST.I, in2 := 28)
      R_Coil( "DBVALVES"."ST6 HOLDFAST LH1".test.fp_HP )
      R_Coil( "DBVALVES"."ST6 HOLDFAST LH1".test.fp_WP )
      R_Coil( "DBVALVES"."ST6 HOLDFAST LH1".test.fp_IDLE )
   END_RUNG
   // the same network as SCL:
   "TEST"(in_nr := 28, out := "DBVALVES"."ST6 HOLDFAST LH1".test);
   IF "FLAGS".TEST.I <> 28 THEN
       "DBVALVES"."ST6 HOLDFAST LH1".test.fp_HP := FALSE;
       "DBVALVES"."ST6 HOLDFAST LH1".test.fp_WP := FALSE;
       "DBVALVES"."ST6 HOLDFAST LH1".test.fp_IDLE := FALSE;
   END_IF;
END_REGION

REGION Network 196: TEST - [29] ST6 HOLDFAST LH2
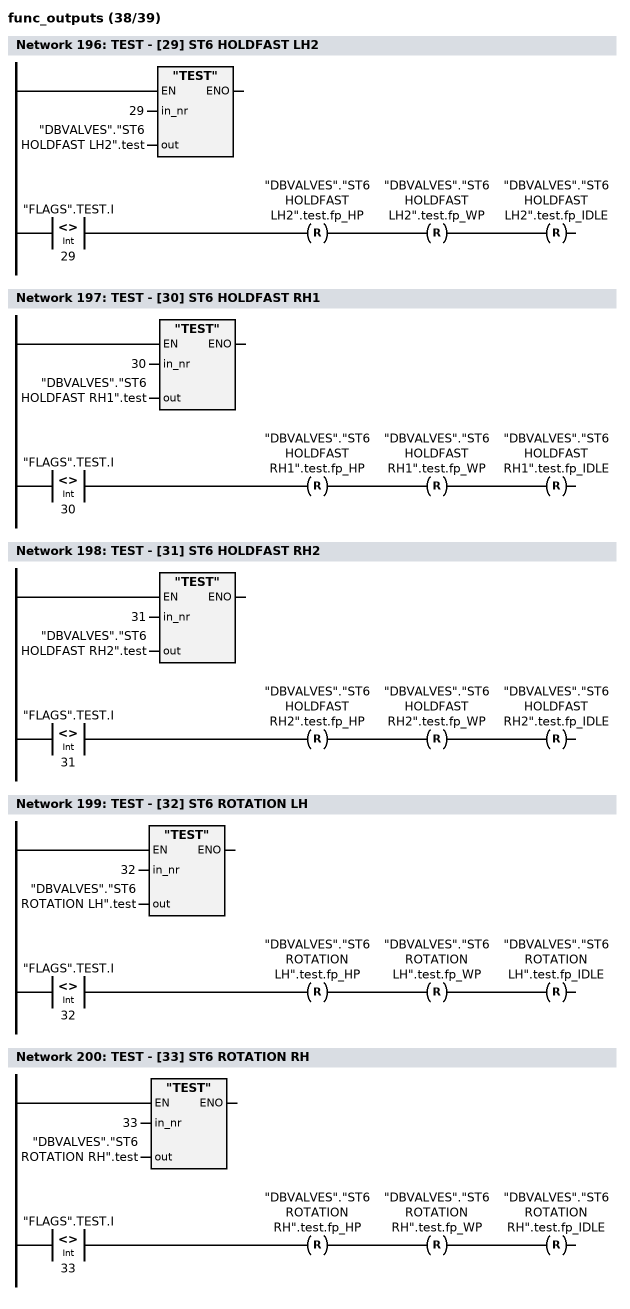
   RUNG wire#powerrail
      "TEST"(in_nr := 29, out := "DBVALVES"."ST6 HOLDFAST LH2".test)
   END_RUNG
   RUNG wire#powerrail
      { S7_Templates := "SrcType := Int" } NE_Contact(in1 := "FLAGS".TEST.I, in2 := 29)
      R_Coil( "DBVALVES"."ST6 HOLDFAST LH2".test.fp_HP )
      R_Coil( "DBVALVES"."ST6 HOLDFAST LH2".test.fp_WP )
      R_Coil( "DBVALVES"."ST6 HOLDFAST LH2".test.fp_IDLE )
   END_RUNG
   // the same network as SCL:
   "TEST"(in_nr := 29, out := "DBVALVES"."ST6 HOLDFAST LH2".test);
   IF "FLAGS".TEST.I <> 29 THEN
       "DBVALVES"."ST6 HOLDFAST LH2".test.fp_HP := FALSE;
       "DBVALVES"."ST6 HOLDFAST LH2".test.fp_WP := FALSE;
       "DBVALVES"."ST6 HOLDFAST LH2".test.fp_IDLE := FALSE;
   END_IF;
END_REGION

REGION Network 197: TEST - [30] ST6 HOLDFAST RH1
   RUNG wire#powerrail
      "TEST"(in_nr := 30, out := "DBVALVES"."ST6 HOLDFAST RH1".test)
   END_RUNG
   RUNG wire#powerrail
      { S7_Templates := "SrcType := Int" } NE_Contact(in1 := "FLAGS".TEST.I, in2 := 30)
      R_Coil( "DBVALVES"."ST6 HOLDFAST RH1".test.fp_HP )
      R_Coil( "DBVALVES"."ST6 HOLDFAST RH1".test.fp_WP )
      R_Coil( "DBVALVES"."ST6 HOLDFAST RH1".test.fp_IDLE )
   END_RUNG
   // the same network as SCL:
   "TEST"(in_nr := 30, out := "DBVALVES"."ST6 HOLDFAST RH1".test);
   IF "FLAGS".TEST.I <> 30 THEN
       "DBVALVES"."ST6 HOLDFAST RH1".test.fp_HP := FALSE;
       "DBVALVES"."ST6 HOLDFAST RH1".test.fp_WP := FALSE;
       "DBVALVES"."ST6 HOLDFAST RH1".test.fp_IDLE := FALSE;
   END_IF;
END_REGION

REGION Network 198: TEST - [31] ST6 HOLDFAST RH2
   RUNG wire#powerrail
      "TEST"(in_nr := 31, out := "DBVALVES"."ST6 HOLDFAST RH2".test)
   END_RUNG
   RUNG wire#powerrail
      { S7_Templates := "SrcType := Int" } NE_Contact(in1 := "FLAGS".TEST.I, in2 := 31)
      R_Coil( "DBVALVES"."ST6 HOLDFAST RH2".test.fp_HP )
      R_Coil( "DBVALVES"."ST6 HOLDFAST RH2".test.fp_WP )
      R_Coil( "DBVALVES"."ST6 HOLDFAST RH2".test.fp_IDLE )
   END_RUNG
   // the same network as SCL:
   "TEST"(in_nr := 31, out := "DBVALVES"."ST6 HOLDFAST RH2".test);
   IF "FLAGS".TEST.I <> 31 THEN
       "DBVALVES"."ST6 HOLDFAST RH2".test.fp_HP := FALSE;
       "DBVALVES"."ST6 HOLDFAST RH2".test.fp_WP := FALSE;
       "DBVALVES"."ST6 HOLDFAST RH2".test.fp_IDLE := FALSE;
   END_IF;
END_REGION

REGION Network 199: TEST - [32] ST6 ROTATION LH
   RUNG wire#powerrail
      "TEST"(in_nr := 32, out := "DBVALVES"."ST6 ROTATION LH".test)
   END_RUNG
   RUNG wire#powerrail
      { S7_Templates := "SrcType := Int" } NE_Contact(in1 := "FLAGS".TEST.I, in2 := 32)
      R_Coil( "DBVALVES"."ST6 ROTATION LH".test.fp_HP )
      R_Coil( "DBVALVES"."ST6 ROTATION LH".test.fp_WP )
      R_Coil( "DBVALVES"."ST6 ROTATION LH".test.fp_IDLE )
   END_RUNG
   // the same network as SCL:
   "TEST"(in_nr := 32, out := "DBVALVES"."ST6 ROTATION LH".test);
   IF "FLAGS".TEST.I <> 32 THEN
       "DBVALVES"."ST6 ROTATION LH".test.fp_HP := FALSE;
       "DBVALVES"."ST6 ROTATION LH".test.fp_WP := FALSE;
       "DBVALVES"."ST6 ROTATION LH".test.fp_IDLE := FALSE;
   END_IF;
END_REGION

REGION Network 200: TEST - [33] ST6 ROTATION RH
   RUNG wire#powerrail
      "TEST"(in_nr := 33, out := "DBVALVES"."ST6 ROTATION RH".test)
   END_RUNG
   RUNG wire#powerrail
      { S7_Templates := "SrcType := Int" } NE_Contact(in1 := "FLAGS".TEST.I, in2 := 33)
      R_Coil( "DBVALVES"."ST6 ROTATION RH".test.fp_HP )
      R_Coil( "DBVALVES"."ST6 ROTATION RH".test.fp_WP )
      R_Coil( "DBVALVES"."ST6 ROTATION RH".test.fp_IDLE )
   END_RUNG
   // the same network as SCL:
   "TEST"(in_nr := 33, out := "DBVALVES"."ST6 ROTATION RH".test);
   IF "FLAGS".TEST.I <> 33 THEN
       "DBVALVES"."ST6 ROTATION RH".test.fp_HP := FALSE;
       "DBVALVES"."ST6 ROTATION RH".test.fp_WP := FALSE;
       "DBVALVES"."ST6 ROTATION RH".test.fp_IDLE := FALSE;
   END_IF;
END_REGION

REGION Network 201: TEST - LAMPS
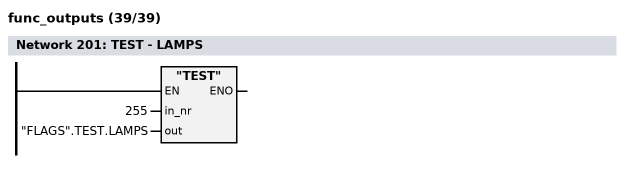
   RUNG wire#powerrail
      "TEST"(in_nr := 255, out := "FLAGS".TEST.LAMPS)
   END_RUNG
   // the same network as SCL:
   "TEST"(in_nr := 255, out := "FLAGS".TEST.LAMPS);
END_REGION
END_FUNCTION
